(* CODESYS project SPT_Components.library
   Company: Beckhoff Automation LLC
   DefaultNamespace: SPT_Components
   Version: 3.1.1
   Placeholder: SPT Components
   Title: SPT Components

Project tree, tasks and I/O mapping:
  libraries: SPT Base Types, * (Beckhoff Automation LLC); SPT Event Logger, * (Beckhoff Automation LLC); SPT Motion Control, * (Beckhoff Automation LLC); SPT Utilities, * (Beckhoff Automation LLC); Tc2_DataExchange, * (Beckhoff Automation GmbH); Tc2_MC2, * (Beckhoff Automation GmbH); Tc2_Standard, * (Beckhoff Automation GmbH); Tc2_System, * (Beckhoff Automation GmbH); Tc3_EventLogger, * (Beckhoff Automation GmbH); Tc3_Module, * (Beckhoff Automation GmbH); TcUnit, * (www.tcunit.org)
  Axes/
    DUT/
      data type ST_AxisBase_Command
      data type ST_AxisBase_Config
      data type ST_AxisBase_HMI
      data type ST_AxisBase_Status
    function block FB_Component_BasicAxis [ST]: Disable, Enable, Home, Jog, MoveAbsolute, MoveModulo, MoveRelative, MoveVelocity, Reset, Stop, WriteBoolParameter, WriteParameter, Acceleration, Deceleration, Jerk, Velocity, ActualAcceleration, ActualPosition, ActualPositionModulo, ActualTorque, ActualVelocity, PositionLag, SetAcceleration, SetPosition, SetPositionModulo, SetVelocity, Enabled, InPosition, Stopped, Axis, HomeMethod, InhibitFeedNegative, InhibitFeedPositive, Override, ResetMethod, CreateEvents, HMICommunication, Monitoring, CyclicLogic, Initialize
    function block FB_Component_BasicSlaveAxis [ST]: Disable, Enable, Home, Jog, MoveAbsolute, MoveModulo, MoveRelative, MoveVelocity, Reset, Stop, WriteBoolParameter, WriteParameter, Acceleration, Deceleration, Jerk, Velocity, ActualAcceleration, ActualPosition, ActualPositionModulo, ActualTorque, ActualVelocity, PositionLag, SetAcceleration, SetPosition, SetPositionModulo, SetVelocity, Enabled, InPosition, Stopped, Axis, HomeMethod, InhibitFeedNegative, InhibitFeedPositive, Override, ResetMethod, GearIn, GearOut, InGear, Master1, Master2, Master3, Master4, RatioMaster1, RatioMaster2, RatioMaster3, RatioMaster4, CreateEvents, HMICommunication, Monitoring, CyclicLogic, Initialize
    function block FB_Component_CamSlaveAxis [ST]: Disable, Enable, Home, Jog, MoveAbsolute, MoveModulo, MoveRelative, MoveVelocity, Reset, Stop, WriteBoolParameter, WriteParameter, Acceleration, Deceleration, Jerk, Velocity, ActualAcceleration, ActualPosition, ActualPositionModulo, ActualTorque, ActualVelocity, PositionLag, SetAcceleration, SetPosition, SetPositionModulo, SetVelocity, Enabled, InPosition, Stopped, Axis, HomeMethod, InhibitFeedNegative, InhibitFeedPositive, Override, ResetMethod, CamParameters, ChangeMode, FindSlavePos, FindSyncPos, InSync, Master, RunningTable, StartCouple, StartSync, SyncPos, UpdateTable, CreateEvents, HMICommunication, Monitoring, CyclicLogic, Initialize
  GVLs/
    global variables CONSTANTS
  Project Information/
    function F_GetCompany [ST]
    function F_GetTitle [ST]
    function F_GetVersion [ST]
  Sensors/
    DUT/
      data type E_DebounceMode
      data type E_SensorSimulationMode
      data type ST_DigitalSensor_Command
      data type ST_DigitalSensor_Config
      data type ST_DigitalSensor_HMI
      data type ST_DigitalSensor_Status
    function block FB_DigitalSensor [ST]: CyclicLogic, Active, DebounceMode, DebounceTime, Inverted, SimulationInput, SimulationMode, SimulationTimeBase, TimeActive, TimeInactive, HMICommunication, Monitoring, ProcessInput
    interface I_DigitalSensorBase: DebounceMode, DebounceTime, Inverted, SimulationInput, SimulationMode, TimeActive, TimeInactive
  Solenoids/
    DUT/
      data type ST_Cylinder_Command
      data type ST_Cylinder_Config
      data type ST_Cylinder_HMI
      data type ST_Cylinder_Status
    SolenoidBankBase/
      data type E_SolenoidType
      function block FB_SolenoidBankBase [ST]: AddSolenoid, CheckNumber, CreateEvents, CyclicLogic, Initialize, MapIO, Monitoring, Reset
      data type ST_SolenoidBankConfig
    function block FB_DoubleSolenoid [ST]: HardwareInit, HardwareUpdate, RetractOutput
    function block FB_DoubleSolenoidFeedback [ST]: ExtendedInput, Feedback, HardwareInit, RetractedInput
    function block FB_SingleSolenoid [ST]: CreateEvents, HMICommunication, Monitoring, CyclicLogic, Extend, Extended, ExtendOutput, ExtendTime, Retract, Retracted, RetractOutput, RetractTime, Feedback, HardwareInit, HardwareUpdate, Initialize, Reset
    function block FB_SingleSolenoidFeedback [ST]: ExtendedInput, Feedback, HardwareInit, RetractedInput
    interface I_Solenoid: Extend, Extended, ExtendOutput, ExtendTime, Retract, Retracted, RetractOutput, RetractTime
    global variables Parameters_Cylinder
  Testing/
    Axis/
      function block FB_ComponentBasicAxis_Test [ST]: AllowHMI, BlockHMI, Busy, CommandInhibited, Init, MCHaltAlarm, MCHomeAlarm, MCJogAlarm, MCMoveAbsoluteAlarm, MCMoveModulo, MCMoveRelativeAlarm, MCMoveVelocity, MCPowerAlarm, McReadAxisParametersAlarm, MCResetAlarm, McWriteAxisBoolParameterAlarm, McWriteAxisParameterAlarm, NameSetProperty, SimulationCheckAlarm, SimulationSetHMI, SimulationSetProperty
    Solenoids/
      function block FB_DoubleSolenoid_Test [ST]: ExtendEqualsExtendOutputOnRetractOff, RetractEqualsExtendOutputOffRetractOutputOn
      function block FB_SingleSolenoid_Test [ST]: AllowHMI, BlockHMI, Busy, ExtendEqualsExtendedOutputOn, Init, NameSetProperty, RetractEqualsExtendOutputOff, SimulationCheckAlarm, SimulationSetHMI, SimulationSetProperty
      function block FB_SingleSolenoidFeedback_Test [ST]: Extend, ExtendError
    global variables GVL_Testing
    program PRG_TEST [ST]
  Version/
    global variables Global_Version
*)

// Axes/DUT/ST_AxisBase_Command
TYPE ST_AxisBase_Command :
	STRUCT
		JogFast_Forward	 : BOOL;
		JogFast_Backward : BOOL;
		JogSlow_Forward	 : BOOL;
		JogSlow_Backward : BOOL;
	END_STRUCT
END_TYPE

// Axes/DUT/ST_AxisBase_Config
TYPE ST_AxisBase_Config :
	STRUCT
		JogFastVelocity : LREAL;
		JogSlowVelocity : LREAL;
	END_STRUCT
END_TYPE

// Axes/DUT/ST_AxisBase_HMI
TYPE ST_AxisBase_HMI :
	STRUCT
		Config	: ST_AxisBase_Config;
		Command : ST_AxisBase_Command;
		Status	: ST_AxisBase_Status;
	END_STRUCT
END_TYPE

// Axes/DUT/ST_AxisBase_Status
TYPE ST_AxisBase_Status :
	STRUCT
		Enabled				 : BOOL;
		InPosition			 : BOOL;
		Stopped				 : BOOL;
		Coupled				 : BOOL;
		SetPosition			 : LREAL;
		SetPositionModulo	 : LREAL;
		SetVelocity			 : LREAL;
		SetAcceleration		 : LREAL;
		ActualPosition		 : LREAL;
		ActualPositionModulo : LREAL;
		ActualVelocity		 : LREAL;
		ActualAcceleration	 : LREAL;
		ActualTorque		 : LREAL;
		PositionLag			 : LREAL;
	END_STRUCT
END_TYPE

// Sensors/DUT/E_DebounceMode
{attribute 'qualified_only'}
{attribute 'strict'}
TYPE E_DebounceMode : (
		RawInput,
		SimpleFlickerFilter,
		EdgeDetectFilter,
		MovingAverage
	) DINT;
END_TYPE

// Sensors/DUT/E_SensorSimulationMode
{attribute 'qualified_only'}
{attribute 'strict'}
TYPE E_SensorSimulationMode : (
		InputDriven, //Follows the state of the SimulationInput property
		Periodic	 //Follows a 50% duty cycle at the period specified in ms by SimulationInput);
	);
END_TYPE

// Sensors/DUT/ST_DigitalSensor_Command
TYPE ST_DigitalSensor_Command :
	STRUCT
	END_STRUCT
END_TYPE

// Sensors/DUT/ST_DigitalSensor_Config
TYPE ST_DigitalSensor_Config :
	STRUCT
		//Status information
		DebounceMode	   : E_DebounceMode;
		DebounceTime	   : TIME;
		Inverted		   : BOOL;
		SimulationMode	   : E_SensorSimulationMode;
		SimulationTimebase : UINT;
	END_STRUCT
END_TYPE

// Sensors/DUT/ST_DigitalSensor_HMI
TYPE ST_DigitalSensor_HMI :
	STRUCT
		Config	: ST_DigitalSensor_Config;
		Command : ST_DigitalSensor_Command;
		Status	: ST_DigitalSensor_Status;
	END_STRUCT
END_TYPE

// Sensors/DUT/ST_DigitalSensor_Status
TYPE ST_DigitalSensor_Status :
	STRUCT
		Active		 : BOOL;
		TimeActive	 : LREAL;
		TimeInactive : LREAL;
	END_STRUCT
END_TYPE

// Solenoids/DUT/ST_Cylinder_Command
TYPE ST_Cylinder_Command :
	STRUCT
		Extend		: BOOL;
		Retract		: BOOL;
		ExtendTime	: LREAL;
		RetractTime : LREAL;
	END_STRUCT
END_TYPE

// Solenoids/DUT/ST_Cylinder_Config
TYPE ST_Cylinder_Config :
	STRUCT
		ExtendTime	: LREAL;
		RetractTime : LREAL;
	END_STRUCT
END_TYPE

// Solenoids/DUT/ST_Cylinder_HMI
TYPE ST_Cylinder_HMI :
	STRUCT
		Config	: ST_Cylinder_Config;
		Command : ST_Cylinder_Command;
		Status	: ST_Cylinder_Status;
	END_STRUCT
END_TYPE

// Solenoids/DUT/ST_Cylinder_Status
TYPE ST_Cylinder_Status :
	STRUCT
		Extended   : BOOL;
		Retracted  : BOOL;
		Extending  : BOOL;
		Retracting : BOOL;
	END_STRUCT
END_TYPE

// Solenoids/SolenoidBankBase/E_SolenoidType
{attribute 'qualified_only'}
{attribute 'strict'}
TYPE E_SolenoidType : (
		Single,
		Double,
		SingleFeedback,
		DoubleFeedback
	);
END_TYPE

// Solenoids/SolenoidBankBase/ST_SolenoidBankConfig
TYPE ST_SolenoidBankConfig :
	STRUCT
		SolenoidType		 : E_SolenoidType;
		ipSolenoid			 : I_Solenoid;
		SolenoidOutputNumber : UINT;
	END_STRUCT
END_TYPE

// GVLs/CONSTANTS
{attribute 'qualified_only'}
VAR_GLOBAL CONSTANT
	BASIC_AXIS_ALARM_COUNT		 : UINT := 17;
	BASIC_SLAVE_AXIS_ALARM_COUNT : UINT := 3;
	CAM_SLAVE_AXIS_ALARM_COUNT	 : UINT := 9;
END_VAR

// Solenoids/Parameters_Cylinder
{attribute 'qualified_only'}
VAR_GLOBAL CONSTANT
	MAX_NUMBER_OF_SOLENOIDS : UINT := 32;
END_VAR

// Testing/GVL_Testing
{attribute 'qualified_only'}
VAR_GLOBAL
	SingleSolenoidTestsDone : BOOL;
END_VAR

// Version/Global_Version
{attribute 'TcGenerated'}
{attribute 'no-analysis'}
{attribute 'linkalways'}
// This function has been automatically generated from the project information.
VAR_GLOBAL CONSTANT
	{attribute 'const_non_replaced'}
	stLibVersion_SPT_Components : ST_LibVersion := (iMajor := 3, iMinor := 1, iBuild := 1, iRevision := 0, nFlags := 1, sVersion := '3.1.1');
END_VAR

// Axes/FB_Component_BasicAxis
FUNCTION_BLOCK FB_Component_BasicAxis EXTENDS FB_ComponentBase IMPLEMENTS I_BasicAxis
VAR
	BasicAxis				: FB_BasicAxis;
	AxisBase_HMI			: ST_AxisBase_HMI;
	BasicAxisAlarms			: ARRAY[1..CONSTANTS.BASIC_AXIS_ALARM_COUNT] OF FB_TcAlarm;
	HMICommand_BasicAxis_RT : R_TRIG;
END_VAR

// There should be no code in the function block body of I_CyclicFB

METHOD Disable : BOOL
Disable := BasicAxis.Disable();
END_METHOD

METHOD Enable : BOOL
Enable := BasicAxis.Enable();
END_METHOD

METHOD Home : BOOL
Home := BasicAxis.Home();
END_METHOD

METHOD Jog : BOOL
VAR_INPUT
	JogFW	 : BOOL;
	JogBW	 : BOOL;
	JogMode	 : E_JogMode;
	Position : LREAL;
END_VAR
Jog := BasicAxis.Jog(JogFW,
					 JogBW,
					 JogMode,
					 Position);
END_METHOD

METHOD MoveAbsolute : BOOL
VAR_INPUT
	Position	  : LREAL;
	AbortPrevious : BOOL;
END_VAR
MoveAbsolute := BasicAxis.MoveAbsolute(Position, AbortPrevious);
END_METHOD

METHOD MoveModulo : BOOL
VAR_INPUT
	Position	  : LREAL;
	Direction	  : MC_Direction;
	AbortPrevious : BOOL;
END_VAR
MoveModulo := BasicAxis.MoveModulo(Position, Direction, AbortPrevious);
END_METHOD

METHOD MoveRelative : BOOL
VAR_INPUT
	Distance	  : LREAL;
	AbortPrevious : BOOL;
END_VAR
MoveRelative := BasicAxis.MoveRelative(Distance, AbortPrevious);
END_METHOD

METHOD MoveVelocity : BOOL
VAR_INPUT
	Velocity	  : LREAL;
	AbortPrevious : BOOL;
END_VAR
MoveVelocity := BasicAxis.MoveVelocity(Velocity, AbortPrevious);
END_METHOD

METHOD Reset : BOOL
Reset := FALSE;
SUPER^.Reset();
IF BasicAxis.ResetMethod = 0 THEN
	RETURN;
ELSIF BasicAxis.HomeMethod = 0 THEN
	RETURN;
ELSE
	IF (BasicAxis.ResetMethod.Error AND BasicAxis.ResetPreviouslyErrored) AND BasicAxisAlarms[E_BasicAxis.ResetError].bRaised THEN
		BasicAxisAlarms[E_BasicAxis.ResetError].Clear(0, 0);
	END_IF

	IF (BasicAxis.HomeMethod.Error AND BasicAxis.HomePreviouslyErrored) AND BasicAxisAlarms[E_BasicAxis.HomeError].bRaised THEN
		BasicAxisAlarms[E_BasicAxis.HomeError].Clear(0, 0);
	END_IF

	IF BasicAxis.Reset() THEN
		_Error	 := FALSE;
		_ErrorID := 0;
		Reset	 := TRUE;
	END_IF
END_IF
END_METHOD

METHOD Stop : BOOL
Stop := BasicAxis.Stop();
END_METHOD

METHOD WriteBoolParameter : BOOL
VAR_INPUT
	ParameterNumber : MC_AxisParameter;
	Value			: BOOL;
END_VAR
WriteBoolParameter := BasicAxis.WriteBoolParameter(ParameterNumber, Value);
END_METHOD

METHOD WriteParameter : BOOL
VAR_INPUT
	ParameterNumber : MC_AxisParameter;
	Value			: LREAL;
END_VAR
WriteParameter := BasicAxis.WriteParameter(ParameterNumber, Value);
END_METHOD

PROPERTY Acceleration : LREAL
GET
Acceleration := BasicAxis.Acceleration;
END_GET
SET
BasicAxis.Acceleration := Acceleration;
END_SET
END_PROPERTY

PROPERTY Deceleration : LREAL
GET
Deceleration := BasicAxis.Deceleration;
END_GET
SET
BasicAxis.Deceleration := Deceleration;
END_SET
END_PROPERTY

PROPERTY Jerk : LREAL
GET
Jerk := BasicAxis.Jerk;
END_GET
SET
BasicAxis.Jerk := Jerk;
END_SET
END_PROPERTY

PROPERTY Velocity : LREAL
GET
Velocity := BasicAxis.Velocity;
END_GET
SET
BasicAxis.Velocity := Velocity;
END_SET
END_PROPERTY

PROPERTY ActualAcceleration : LREAL
GET
ActualAcceleration := BasicAxis.ActualAcceleration;
END_GET
END_PROPERTY

PROPERTY ActualPosition : LREAL
GET
ActualPosition := BasicAxis.ActualPosition;
END_GET
END_PROPERTY

PROPERTY ActualPositionModulo : LREAL
GET
ActualPositionModulo := BasicAxis.ActualPositionModulo;
END_GET
END_PROPERTY

PROPERTY ActualTorque : LREAL
GET
ActualTorque := BasicAxis.ActualTorque;
END_GET
END_PROPERTY

PROPERTY ActualVelocity : LREAL
GET
ActualVelocity := BasicAxis.ActualVelocity;
END_GET
END_PROPERTY

PROPERTY PositionLag : LREAL
GET
PositionLag := BasicAxis.PositionLag;
END_GET
END_PROPERTY

PROPERTY SetAcceleration : LREAL
GET
SetAcceleration := BasicAxis.SetAcceleration;
END_GET
END_PROPERTY

PROPERTY SetPosition : LREAL
GET
SetPosition := BasicAxis.SetPosition;
END_GET
END_PROPERTY

PROPERTY SetPositionModulo : LREAL
GET
SetPositionModulo := BasicAxis.SetPositionModulo;
END_GET
END_PROPERTY

PROPERTY SetVelocity : LREAL
GET
SetVelocity := BasicAxis.SetVelocity;
END_GET
END_PROPERTY

PROPERTY Enabled : BOOL
GET
Enabled := BasicAxis.Enabled;
END_GET
END_PROPERTY

PROPERTY InPosition : BOOL
GET
InPosition := BasicAxis.InPosition;
END_GET
END_PROPERTY

PROPERTY Stopped : BOOL
GET
Stopped := BasicAxis.Stopped;
END_GET
END_PROPERTY

{attribute 'analysis' := '-29'}
PROPERTY Axis : REFERENCE TO AXIS_REF
GET
Axis REF= BasicAxis.Axis;
END_GET
END_PROPERTY

PROPERTY HomeMethod : I_MotionSequence
SET
BasicAxis.HomeMethod := HomeMethod;
END_SET
END_PROPERTY

PROPERTY InhibitFeedNegative : BOOL
SET
BasicAxis.InhibitFeedNegative := InhibitFeedNegative;
END_SET
END_PROPERTY

PROPERTY InhibitFeedPositive : BOOL
SET
BasicAxis.InhibitFeedPositive := InhibitFeedPositive;
END_SET
END_PROPERTY

PROPERTY Override : LREAL
GET
Override := BasicAxis.Override;
END_GET
SET
IF Override >= 0 AND Override <= 100 THEN
	BasicAxis.Override := Override;
END_IF
END_SET
END_PROPERTY

PROPERTY ResetMethod : I_MotionSequence
SET
BasicAxis.ResetMethod := ResetMethod;
END_SET
END_PROPERTY

{attribute 'call_after_online_change_slot' := '<slot>'}
METHOD PROTECTED CreateEvents
VAR
	Temp : STRING;
END_VAR
Temp := CONCAT(CONCAT(CONCAT('Axis ', ': '), Name),
			   ' '); //Creates a utility string for alarms and other messaging that reads (example text) - "Module 10 - Main Casepacker" to be followed by the alarm or message info

F_CreateAllEventsInClass(Alarms		:= BasicAxisAlarms,
						 ClassSize	:= SIZEOF(TC_EVENTS.BasicAxis),
						 pInitEvent := ADR(TC_EVENTS.BasicAxis.InitReferenceEvent),
						 Prefix		:= Name);

SUPER^.CreateEvents();
END_METHOD

METHOD PROTECTED HMICommunication
//Extend this method in extended FBs to communicate specific implementation data
SUPER^.HMICommunication();

//Process HMI requests

//Replace 'FALSE' below with further momentary commands (myCommand XOR myOtherCommand XOR...)
HMICommand_BasicAxis_RT(CLK := (ComponentBase_HMI.Status.HMIControlAvailable AND NOT HMICommandActive_Base));

//Signal to FB_ComponentBase that a command is active
HMICommandActive_Descendant := ComponentBase_HMI.Status.HMIControlAvailable AND
							   (AxisBase_HMI.Command.JogFast_Backward OR AxisBase_HMI.Command.JogFast_Forward OR AxisBase_HMI.Command.JogSlow_Forward OR AxisBase_HMI.Command.JogSlow_Backward);

//Process HMI requests
IF HMICommand_BasicAxis_RT.Q THEN //If a request has been issued by the HMI, and a previous request has not just finished being processed
END_IF

IF ComponentBase_HMI.Status.HMIControlAvailable AND NOT HMICommand_BasicAxis_RT.Q THEN
	IF AxisBase_HMI.Command.JogSlow_Forward THEN
		BasicAxis.Jog(AxisBase_HMI.Command.JogSlow_Forward,
					  FALSE,
					  E_JogMode.MC_JOGMODE_STANDARD_SLOW,
					  0.0);
	ELSIF AxisBase_HMI.Command.JogSlow_Backward THEN
		BasicAxis.Jog(FALSE,
					  AxisBase_HMI.Command.JogSlow_Backward,
					  E_JogMode.MC_JOGMODE_STANDARD_SLOW,
					  0.0);
	ELSIF AxisBase_HMI.Command.JogFast_Forward THEN
		BasicAxis.Jog(AxisBase_HMI.Command.JogFast_Forward,
					  FALSE,
					  E_JogMode.MC_JOGMODE_STANDARD_FAST,
					  0.0);
	ELSIF AxisBase_HMI.Command.JogFast_Backward THEN
		BasicAxis.Jog(FALSE,
					  AxisBase_HMI.Command.JogFast_Backward,
					  E_JogMode.MC_JOGMODE_STANDARD_FAST,
					  0.0);
	ELSE
		BasicAxis.Jog(FALSE,
					  FALSE,
					  E_JogMode.MC_JOGMODE_STANDARD_SLOW,
					  0.0);
	END_IF
END_IF

//Update HMI status info
AxisBase_HMI.Status.Enabled				 := BasicAxis.Enabled;
AxisBase_HMI.Status.InPosition			 := BasicAxis.InPosition;
AxisBase_HMI.Status.Stopped				 := BasicAxis.Stopped;
AxisBase_HMI.Status.Coupled				 := FALSE;
AxisBase_HMI.Status.SetPosition			 := BasicAxis.SetPosition;
AxisBase_HMI.Status.SetPositionModulo	 := BasicAxis.SetPositionModulo;
AxisBase_HMI.Status.SetVelocity			 := BasicAxis.SetVelocity;
AxisBase_HMI.Status.SetAcceleration		 := BasicAxis.SetAcceleration;
AxisBase_HMI.Status.ActualPosition		 := BasicAxis.ActualPosition;
AxisBase_HMI.Status.ActualPositionModulo := BasicAxis.ActualPositionModulo;
AxisBase_HMI.Status.ActualVelocity		 := BasicAxis.ActualVelocity;
AxisBase_HMI.Status.ActualAcceleration	 := BasicAxis.ActualAcceleration;
AxisBase_HMI.Status.ActualTorque		 := BasicAxis.ActualTorque;
AxisBase_HMI.Status.PositionLag			 := BasicAxis.PositionLag;
END_METHOD

METHOD PROTECTED Monitoring
SUPER^.Monitoring();

//ErrorID 2 - MC_Power
IF BasicAxis.MCPower.Error AND NOT BasicAxisAlarms[E_BasicAxis.PowerError].bRaised THEN
	RaiseAlarmWithStrings(Alarm := BasicAxisAlarms[E_BasicAxis.PowerError], UDINT_TO_STRING(BasicAxis.ErrorID), '');
ELSIF NOT BasicAxis.MCPower.Error AND BasicAxisAlarms[E_BasicAxis.PowerError].bRaised THEN
	BasicAxisAlarms[E_BasicAxis.PowerError].Clear(0, 0);
END_IF

//ErrorID 3 - MC_Reset (or other reset method)
IF BasicAxis.ResetMethod <> 0 THEN
	IF (BasicAxis.ResetMethod.Error AND NOT BasicAxis.ResetPreviouslyErrored) AND NOT BasicAxisAlarms[E_BasicAxis.ResetError].bRaised THEN
		RaiseAlarmWithStrings(Alarm := BasicAxisAlarms[E_BasicAxis.ResetError], UDINT_TO_STRING(BasicAxis.ResetMethod.ErrorID), '');
	ELSIF NOT BasicAxis.ResetMethod.Error AND BasicAxisAlarms[E_BasicAxis.ResetError].bRaised THEN
		BasicAxisAlarms[E_BasicAxis.ResetError].Clear(0, 0);
	END_IF
END_IF

//ErrorID 4 - MC_Halt
IF BasicAxis.MCHalt.Error AND NOT BasicAxisAlarms[E_BasicAxis.HaltError].bRaised THEN
	RaiseAlarmWithStrings(Alarm := BasicAxisAlarms[E_BasicAxis.HaltError], UDINT_TO_STRING(BasicAxis.MCHalt.ErrorID), '');
ELSIF NOT BasicAxis.MCHalt.Error AND BasicAxisAlarms[E_BasicAxis.HaltError].bRaised THEN
	BasicAxisAlarms[E_BasicAxis.HaltError].Clear(0, 0);
END_IF

//ErrorID 5 - MC_Stop **NOT IMPLEMENTED**

//ErrorID 6 - MC_Home (or other home method)
IF BasicAxis.HomeMethod <> 0 THEN
	IF (BasicAxis.HomeMethod.Error AND NOT BasicAxis.HomePreviouslyErrored) AND NOT BasicAxisAlarms[E_BasicAxis.HomeError].bRaised THEN
		RaiseAlarmWithStrings(Alarm := BasicAxisAlarms[E_BasicAxis.HomeError], UDINT_TO_STRING(BasicAxis.HomeMethod.ErrorID), '');
	ELSIF NOT BasicAxis.HomeMethod.Error AND BasicAxisAlarms[E_BasicAxis.HomeError].bRaised THEN
		BasicAxisAlarms[E_BasicAxis.HomeError].Clear(0, 0);
	END_IF
END_IF

//ErrorID 7 - MC_Jog 
IF BasicAxis.MCJog.Error AND NOT BasicAxisAlarms[E_BasicAxis.JogError].bRaised THEN
	RaiseAlarmWithStrings(Alarm := BasicAxisAlarms[E_BasicAxis.JogError], UDINT_TO_STRING(BasicAxis.MCJog.ErrorID), '');
ELSIF NOT BasicAxis.MCJog.Error AND BasicAxisAlarms[E_BasicAxis.JogError].bRaised THEN
	BasicAxisAlarms[E_BasicAxis.JogError].Clear(0, 0);
END_IF

//ErrorID 8 - MC_MoveAbsolute
IF BasicAxis.MCMoveAbsolute <> 0 THEN
	IF BasicAxis.MCMoveAbsolute^.Error AND NOT BasicAxisAlarms[E_BasicAxis.MoveAbsoluteError].bRaised THEN
		RaiseAlarmWithStrings(Alarm := BasicAxisAlarms[E_BasicAxis.MoveAbsoluteError], UDINT_TO_STRING(BasicAxis.MCMoveAbsolute^.ErrorID), '');
	ELSIF NOT BasicAxis.MCMoveAbsolute^.Error AND BasicAxisAlarms[E_BasicAxis.MoveAbsoluteError].bRaised THEN
		BasicAxisAlarms[E_BasicAxis.MoveAbsoluteError].Clear(0, 0);
	END_IF
END_IF

//ErrorID 9 - MC_MoveRelative
IF BasicAxis.MCMoveRelative <> 0 THEN
	IF BasicAxis.MCMoveRelative^.Error AND NOT BasicAxisAlarms[E_BasicAxis.MoveRelativeError].bRaised THEN
		RaiseAlarmWithStrings(Alarm := BasicAxisAlarms[E_BasicAxis.MoveRelativeError], UDINT_TO_STRING(BasicAxis.MCMoveRelative^.ErrorID), '');
	ELSIF NOT BasicAxis.MCMoveRelative^.Error AND BasicAxisAlarms[E_BasicAxis.MoveRelativeError].bRaised THEN
		BasicAxisAlarms[E_BasicAxis.MoveRelativeError].Clear(0, 0);
	END_IF
END_IF

//ErrorID 10 - MC_MoveVelocity
IF BasicAxis.MCMoveVelocity <> 0 THEN
	IF BasicAxis.MCMoveVelocity^.Error AND NOT BasicAxisAlarms[E_BasicAxis.MoveVelocityError].bRaised THEN
		RaiseAlarmWithStrings(Alarm := BasicAxisAlarms[E_BasicAxis.MoveVelocityError], UDINT_TO_STRING(BasicAxis.MCMoveVelocity^.ErrorID), '');
	ELSIF NOT BasicAxis.MCMoveVelocity^.Error AND BasicAxisAlarms[E_BasicAxis.MoveVelocityError].bRaised THEN
		BasicAxisAlarms[E_BasicAxis.MoveVelocityError].Clear(0, 0);
	END_IF
END_IF

//ErrorID 11 - MC_MoveModulo
IF BasicAxis.MCMoveModulo <> 0 THEN
	IF BasicAxis.MCMoveModulo^.Error AND NOT BasicAxisAlarms[E_BasicAxis.MoveModuloError].bRaised THEN
		RaiseAlarmWithStrings(Alarm := BasicAxisAlarms[E_BasicAxis.MoveModuloError], UDINT_TO_STRING(BasicAxis.MCMoveModulo^.ErrorID), '');
	ELSIF NOT BasicAxis.MCMoveModulo^.Error AND BasicAxisAlarms[E_BasicAxis.MoveModuloError].bRaised THEN
		BasicAxisAlarms[E_BasicAxis.MoveModuloError].Clear(0, 0);
	END_IF
END_IF

//ErrorID 12 - MC_ReadParameterSet
IF BasicAxis.MCReadParameterSet.Error AND NOT BasicAxisAlarms[E_BasicAxis.ReadParameterSetError].bRaised THEN
	RaiseAlarmWithStrings(Alarm := BasicAxisAlarms[E_BasicAxis.ReadParameterSetError], UDINT_TO_STRING(BasicAxis.MCReadParameterSet.ErrorID), '');
ELSIF NOT BasicAxis.MCReadParameterSet.Error AND BasicAxisAlarms[E_BasicAxis.ReadParameterSetError].bRaised THEN
	BasicAxisAlarms[E_BasicAxis.ReadParameterSetError].Clear(0, 0);
END_IF

//ErrorID 13 - MC_WriteParameter
IF BasicAxis.MCWriteParameter.Error AND NOT BasicAxisAlarms[E_BasicAxis.WriteParameterError].bRaised THEN
	RaiseAlarmWithStrings(Alarm := BasicAxisAlarms[E_BasicAxis.WriteParameterError], UDINT_TO_STRING(BasicAxis.MCWriteParameter.ErrorID), '');
ELSIF NOT BasicAxis.MCWriteParameter.Error AND BasicAxisAlarms[E_BasicAxis.WriteParameterError].bRaised THEN
	BasicAxisAlarms[E_BasicAxis.WriteParameterError].Clear(0, 0);
END_IF

//ErrorID 14 - MC_WriteBoolParameter
IF BasicAxis.MCWriteBoolParameter.Error AND NOT BasicAxisAlarms[E_BasicAxis.WriteBoolParameterError].bRaised THEN
	RaiseAlarmWithStrings(Alarm := BasicAxisAlarms[E_BasicAxis.WriteBoolParameterError], UDINT_TO_STRING(BasicAxis.MCWriteBoolParameter.ErrorID), '');
ELSIF NOT BasicAxis.MCWriteBoolParameter.Error AND BasicAxisAlarms[E_BasicAxis.WriteBoolParameterError].bRaised THEN
	BasicAxisAlarms[E_BasicAxis.WriteBoolParameterError].Clear(0, 0);
END_IF

//ErrorID 15 - Command While Inhibited (WARNING)
IF ((BasicAxis.Override <= 0) AND _Busy) AND NOT BasicAxisAlarms[E_BasicAxis.CommandWhileInhibited].bRaised THEN
	RaiseAlarm(Alarm := BasicAxisAlarms[E_BasicAxis.CommandWhileInhibited]);
ELSIF NOT ((BasicAxis.Override <= 0) AND _Busy) AND BasicAxisAlarms[E_BasicAxis.CommandWhileInhibited].bRaised THEN
	BasicAxisAlarms[E_BasicAxis.CommandWhileInhibited].Clear(0, 0);
END_IF

//ErrorID 16 - NC Axis Error
IF BasicAxis.Axis.Status.Error AND NOT BasicAxisAlarms[E_BasicAxis.AxisError].bRaised THEN
	RaiseAlarmWithStrings(Alarm := BasicAxisAlarms[E_BasicAxis.AxisError], UDINT_TO_STRING(BasicAxis.Axis.Status.ErrorID), '');
ELSIF NOT BasicAxis.Axis.Status.Error AND BasicAxisAlarms[E_BasicAxis.AxisError].bRaised THEN
	BasicAxisAlarms[E_BasicAxis.AxisError].Clear(0, 0);
END_IF

//ErrorID 17 - Hardware Error **TODO**
_CurrentAlarmSeverity := F_GetMaxSeverityRaised(Alarms := BasicAxisAlarms, CurrentSeverity := CurrentAlarmSeverity);
END_METHOD

METHOD CyclicLogic
SUPER^.CyclicLogic();
BasicAxis.CyclicLogic();
_Busy	 := BasicAxis.Busy;
_Error	 := BasicAxis.Error;
_ErrorID := BasicAxis.ErrorID;
END_METHOD

//! @summary Basic component initialization logic
METHOD PROTECTED Initialize : BOOL;

//! @description This method is called by <c>CyclicLogic()</c> as required
Initialize := FALSE;
IF NOT BasicAxis.InitComplete THEN
	RETURN;
END_IF

Initialize := SUPER^.Initialize();
END_METHOD

END_FUNCTION_BLOCK

// Axes/FB_Component_BasicSlaveAxis
FUNCTION_BLOCK FB_Component_BasicSlaveAxis EXTENDS FB_ComponentBase IMPLEMENTS I_BasicSlaveAxis
VAR
	BasicSlaveAxis				 : FB_BasicSlaveAxis;
	AxisBase_HMI				 : ST_AxisBase_HMI;
	BasicAxisAlarms				 : ARRAY[1..CONSTANTS.BASIC_AXIS_ALARM_COUNT] OF FB_TcAlarm;
	BasicSlaveAxisAlarms		 : ARRAY[1..CONSTANTS.BASIC_SLAVE_AXIS_ALARM_COUNT] OF FB_TcAlarm;
	HMICommand_BasicSlaveAxis_RT : R_TRIG;
END_VAR

// There should be no code in the function block body of I_CyclicFB

METHOD Disable : BOOL
Disable := BasicSlaveAxis.Disable();
END_METHOD

METHOD Enable : BOOL
Enable := BasicSlaveAxis.Enable();
END_METHOD

METHOD Home : BOOL
Home := BasicSlaveAxis.Home();
END_METHOD

METHOD Jog : BOOL
VAR_INPUT
	JogFW	 : BOOL;
	JogBW	 : BOOL;
	JogMode	 : E_JogMode;
	Position : LREAL;
END_VAR
Jog := BasicSlaveAxis.Jog(JogFW,
						  JogBW,
						  JogMode,
						  Position);
END_METHOD

METHOD MoveAbsolute : BOOL
VAR_INPUT
	Position	  : LREAL;
	AbortPrevious : BOOL;
END_VAR
MoveAbsolute := BasicSlaveAxis.MoveAbsolute(Position, AbortPrevious);
END_METHOD

METHOD MoveModulo : BOOL
VAR_INPUT
	Position	  : LREAL;
	Direction	  : MC_Direction;
	AbortPrevious : BOOL;
END_VAR
MoveModulo := BasicSlaveAxis.MoveModulo(Position, Direction, AbortPrevious);
END_METHOD

METHOD MoveRelative : BOOL
VAR_INPUT
	Distance	  : LREAL;
	AbortPrevious : BOOL;
END_VAR
MoveRelative := BasicSlaveAxis.MoveRelative(Distance, AbortPrevious);
END_METHOD

METHOD MoveVelocity : BOOL
VAR_INPUT
	Velocity	  : LREAL;
	AbortPrevious : BOOL;
END_VAR
MoveVelocity := BasicSlaveAxis.MoveVelocity(Velocity, AbortPrevious);
END_METHOD

METHOD Reset : BOOL
SUPER^.Reset();
IF BasicSlaveAxis.ResetMethod = 0 THEN
	RETURN;
ELSE
	IF (BasicSlaveAxis.ResetMethod.Error AND BasicSlaveAxis.ResetPreviouslyErrored) AND BasicAxisAlarms[E_BasicAxis.ResetError].bRaised THEN
		BasicAxisAlarms[E_BasicAxis.ResetError].Clear(0, 0);
	END_IF

	IF (BasicSlaveAxis.HomeMethod.Error AND BasicSlaveAxis.HomePreviouslyErrored) AND BasicAxisAlarms[E_BasicAxis.HomeError].bRaised THEN
		BasicAxisAlarms[E_BasicAxis.HomeError].Clear(0, 0);
	END_IF

	IF BasicSlaveAxis.Reset() THEN
		_Error	 := FALSE;
		_ErrorID := 0;
		Reset	 := TRUE;
	END_IF
END_IF
END_METHOD

METHOD Stop : BOOL
Stop := BasicSlaveAxis.Stop();
END_METHOD

METHOD WriteBoolParameter : BOOL
VAR_INPUT
	ParameterNumber : MC_AxisParameter;
	Value			: BOOL;
END_VAR
WriteBoolParameter := BasicSlaveAxis.WriteBoolParameter(ParameterNumber, Value);
END_METHOD

METHOD WriteParameter : BOOL
VAR_INPUT
	ParameterNumber : MC_AxisParameter;
	Value			: LREAL;
END_VAR
WriteParameter := BasicSlaveAxis.WriteParameter(ParameterNumber, Value);
END_METHOD

PROPERTY Acceleration : LREAL
GET
Acceleration := BasicSlaveAxis.Acceleration;
END_GET
SET
BasicSlaveAxis.Acceleration := Acceleration;
END_SET
END_PROPERTY

PROPERTY Deceleration : LREAL
GET
Deceleration := BasicSlaveAxis.Deceleration;
END_GET
SET
BasicSlaveAxis.Deceleration := Deceleration;
END_SET
END_PROPERTY

PROPERTY Jerk : LREAL
GET
Jerk := BasicSlaveAxis.Jerk;
END_GET
SET
BasicSlaveAxis.Jerk := Jerk;
END_SET
END_PROPERTY

PROPERTY Velocity : LREAL
GET
Velocity := BasicSlaveAxis.Velocity;
END_GET
SET
BasicSlaveAxis.Velocity := Velocity;
END_SET
END_PROPERTY

PROPERTY ActualAcceleration : LREAL
GET
ActualAcceleration := BasicSlaveAxis.ActualAcceleration;
END_GET
END_PROPERTY

PROPERTY ActualPosition : LREAL
GET
ActualPosition := BasicSlaveAxis.ActualPosition;
END_GET
END_PROPERTY

PROPERTY ActualPositionModulo : LREAL
GET
ActualPositionModulo := BasicSlaveAxis.ActualPositionModulo;
END_GET
END_PROPERTY

PROPERTY ActualTorque : LREAL
GET
ActualTorque := BasicSlaveAxis.ActualTorque;
END_GET
END_PROPERTY

PROPERTY ActualVelocity : LREAL
GET
ActualVelocity := BasicSlaveAxis.ActualVelocity;
END_GET
END_PROPERTY

PROPERTY PositionLag : LREAL
GET
PositionLag := BasicSlaveAxis.PositionLag;
END_GET
END_PROPERTY

PROPERTY SetAcceleration : LREAL
GET
SetAcceleration := BasicSlaveAxis.SetAcceleration;
END_GET
END_PROPERTY

PROPERTY SetPosition : LREAL
GET
SetPosition := BasicSlaveAxis.SetPosition;
END_GET
END_PROPERTY

PROPERTY SetPositionModulo : LREAL
GET
SetPositionModulo := BasicSlaveAxis.SetPositionModulo;
END_GET
END_PROPERTY

PROPERTY SetVelocity : LREAL
GET
SetVelocity := BasicSlaveAxis.SetVelocity;
END_GET
END_PROPERTY

PROPERTY Enabled : BOOL
GET
Enabled := BasicSlaveAxis.Enabled;
END_GET
END_PROPERTY

PROPERTY InPosition : BOOL
GET
InPosition := BasicSlaveAxis.InPosition;
END_GET
END_PROPERTY

PROPERTY Stopped : BOOL
GET
Stopped := BasicSlaveAxis.Stopped;
END_GET
END_PROPERTY

PROPERTY Axis : REFERENCE TO AXIS_REF
GET
Axis REF= BasicSlaveAxis.Axis;
END_GET
END_PROPERTY

PROPERTY HomeMethod : I_MotionSequence
SET
BasicSlaveAxis.HomeMethod := HomeMethod;
END_SET
END_PROPERTY

PROPERTY InhibitFeedNegative : BOOL
SET
BasicSlaveAxis.InhibitFeedNegative := InhibitFeedNegative;
END_SET
END_PROPERTY

PROPERTY InhibitFeedPositive : BOOL
SET
BasicSlaveAxis.InhibitFeedPositive := InhibitFeedPositive;
END_SET
END_PROPERTY

PROPERTY Override : LREAL
GET
Override := BasicSlaveAxis.Override;
END_GET
SET
IF Override >= 0 AND Override <= 100 THEN
	BasicSlaveAxis.Override := Override;
END_IF
END_SET
END_PROPERTY

PROPERTY ResetMethod : I_MotionSequence
SET
BasicSlaveAxis.ResetMethod := ResetMethod;
END_SET
END_PROPERTY

METHOD PUBLIC GearIn : BOOL
VAR_INPUT
END_VAR
GearIn := BasicSlaveAxis.GearIn();
END_METHOD

METHOD GearOut : BOOL
GearOut := BasicSlaveAxis.GearOut();
END_METHOD

PROPERTY InGear : BOOL
GET
InGear := BasicSlaveAxis.InGear;
END_GET
END_PROPERTY

PROPERTY Master1 : REFERENCE TO AXIS_REF
GET
IF __ISVALIDREF(BasicSlaveAxis.Master1) THEN
	Master1 REF= BasicSlaveAxis.Master1;
END_IF
END_GET
SET
BasicSlaveAxis.Master1 REF= Master1;
END_SET
END_PROPERTY

PROPERTY Master2 : REFERENCE TO AXIS_REF
GET
IF __ISVALIDREF(BasicSlaveAxis.Master2) THEN
	Master2 REF= BasicSlaveAxis.Master2;
END_IF
END_GET
SET
BasicSlaveAxis.Master2 REF= Master2;
END_SET
END_PROPERTY

PROPERTY Master3 : REFERENCE TO AXIS_REF
GET
IF __ISVALIDREF(BasicSlaveAxis.Master3) THEN
	Master3 REF= BasicSlaveAxis.Master3;
END_IF
END_GET
SET
BasicSlaveAxis.Master3 REF= Master3;
END_SET
END_PROPERTY

PROPERTY Master4 : REFERENCE TO AXIS_REF
GET
IF __ISVALIDREF(BasicSlaveAxis.Master4) THEN
	Master4 REF= BasicSlaveAxis.Master4;
END_IF
END_GET
SET
BasicSlaveAxis.Master4 REF= Master4;
END_SET
END_PROPERTY

PROPERTY RatioMaster1 : LREAL
GET
RatioMaster1 := BasicSlaveAxis.RatioMaster1;
END_GET
SET
BasicSlaveAxis.RatioMaster1 := RatioMaster1;
END_SET
END_PROPERTY

PROPERTY RatioMaster2 : LREAL
GET
RatioMaster2 := BasicSlaveAxis.RatioMaster2;
END_GET
SET
BasicSlaveAxis.RatioMaster2 := RatioMaster2;
END_SET
END_PROPERTY

PROPERTY RatioMaster3 : LREAL
GET
RatioMaster3 := BasicSlaveAxis.RatioMaster3;
END_GET
SET
BasicSlaveAxis.RatioMaster3 := RatioMaster3;
END_SET
END_PROPERTY

PROPERTY RatioMaster4 : LREAL
GET
RatioMaster4 := BasicSlaveAxis.RatioMaster4;
END_GET
SET
BasicSlaveAxis.RatioMaster4 := RatioMaster4;
END_SET
END_PROPERTY

{attribute 'call_after_online_change_slot' := '<slot>'}
METHOD PROTECTED CreateEvents
VAR
	Temp : STRING;
END_VAR
Temp := CONCAT(CONCAT(CONCAT('Axis ', ': '), Name),
			   ' '); //Creates a utility string for alarms and other messaging that reads (example text) - "Module 10 - Main Casepacker" to be followed by the alarm or message info

F_CreateAllEventsInClass(Alarms		:= BasicAxisAlarms,
						 ClassSize	:= SIZEOF(TC_EVENTS.BasicAxis),
						 pInitEvent := ADR(TC_EVENTS.BasicAxis.InitReferenceEvent),
						 Prefix		:= Name);

F_CreateAllEventsInClass(Alarms		:= BasicSlaveAxisAlarms,
						 ClassSize	:= SIZEOF(TC_EVENTS.BasicSlaveAxis),
						 pInitEvent := ADR(TC_EVENTS.BasicSlaveAxis.InitReferenceEvent),
						 Prefix		:= Name);

SUPER^.CreateEvents();
END_METHOD

METHOD PROTECTED HMICommunication
//Extend this method in extended FBs to communicate specific implementation data
SUPER^.HMICommunication();

//Process HMI requests

//Replace 'FALSE' below with further momentary commands (myCommand XOR myOtherCommand XOR...)
HMICommand_BasicSlaveAxis_RT(CLK := (ComponentBase_HMI.Status.HMIControlAvailable AND NOT HMICommandActive_Base) AND (FALSE));

//Signal to FB_ComponentBase that a command is active
HMICommandActive_Descendant := ComponentBase_HMI.Status.HMIControlAvailable AND
							   (AxisBase_HMI.Command.JogFast_Backward OR AxisBase_HMI.Command.JogFast_Forward OR AxisBase_HMI.Command.JogSlow_Forward OR AxisBase_HMI.Command.JogSlow_Backward);

IF HMICommand_BasicSlaveAxis_RT.Q THEN
	;
END_IF

//Process HMI requests
IF HMICommand_BasicSlaveAxis_RT.Q THEN //If a request has been issued by the HMI, and a previous request has not just finished being processed

	//	IF AxisBaseHMI.Command.xxx THEN

	//		Enabled := TRUE;

	//	END_IF
END_IF

IF ComponentBase_HMI.Status.HMIControlAvailable AND NOT HMICommand_BasicSlaveAxis_RT.Q THEN
	IF AxisBase_HMI.Command.JogSlow_Forward THEN
		BasicSlaveAxis.Jog(AxisBase_HMI.Command.JogSlow_Forward,
						   FALSE,
						   E_JogMode.MC_JOGMODE_STANDARD_SLOW,
						   0.0);
	ELSIF AxisBase_HMI.Command.JogSlow_Backward THEN
		BasicSlaveAxis.Jog(FALSE,
						   AxisBase_HMI.Command.JogSlow_Backward,
						   E_JogMode.MC_JOGMODE_STANDARD_SLOW,
						   0.0);
	ELSIF AxisBase_HMI.Command.JogFast_Forward THEN
		BasicSlaveAxis.Jog(AxisBase_HMI.Command.JogFast_Forward,
						   FALSE,
						   E_JogMode.MC_JOGMODE_STANDARD_FAST,
						   0.0);
	ELSIF AxisBase_HMI.Command.JogFast_Backward THEN
		BasicSlaveAxis.Jog(FALSE,
						   AxisBase_HMI.Command.JogFast_Backward,
						   E_JogMode.MC_JOGMODE_STANDARD_FAST,
						   0.0);
	ELSE
		BasicSlaveAxis.Jog(FALSE,
						   FALSE,
						   E_JogMode.MC_JOGMODE_STANDARD_SLOW,
						   0.0);
	END_IF
END_IF

//Update HMI status info
AxisBase_HMI.Status.Enabled				 := BasicSlaveAxis.Enabled;
AxisBase_HMI.Status.InPosition			 := BasicSlaveAxis.InPosition;
AxisBase_HMI.Status.Stopped				 := BasicSlaveAxis.Stopped;
AxisBase_HMI.Status.Coupled				 := BasicSlaveAxis.InGear;
AxisBase_HMI.Status.SetPosition			 := BasicSlaveAxis.SetPosition;
AxisBase_HMI.Status.SetPositionModulo	 := BasicSlaveAxis.SetPositionModulo;
AxisBase_HMI.Status.SetVelocity			 := BasicSlaveAxis.SetVelocity;
AxisBase_HMI.Status.SetAcceleration		 := BasicSlaveAxis.SetAcceleration;
AxisBase_HMI.Status.ActualPosition		 := BasicSlaveAxis.ActualPosition;
AxisBase_HMI.Status.ActualPositionModulo := BasicSlaveAxis.ActualPositionModulo;
AxisBase_HMI.Status.ActualVelocity		 := BasicSlaveAxis.ActualVelocity;
AxisBase_HMI.Status.ActualAcceleration	 := BasicSlaveAxis.ActualAcceleration;
AxisBase_HMI.Status.ActualTorque		 := BasicSlaveAxis.ActualTorque;
AxisBase_HMI.Status.PositionLag			 := BasicSlaveAxis.PositionLag;
END_METHOD

METHOD PROTECTED Monitoring
SUPER^.Monitoring();

(* Basic Axis Alarms *)

//ErrorID 2 - MC_Power
IF BasicSlaveAxis.MCPower.Error AND NOT BasicAxisAlarms[E_BasicAxis.PowerError].bRaised THEN
	RaiseAlarmWithStrings(Alarm := BasicAxisAlarms[E_BasicAxis.PowerError], UDINT_TO_STRING(BasicSlaveAxis.ErrorID), '');
ELSIF NOT BasicSlaveAxis.MCPower.Error AND BasicAxisAlarms[E_BasicAxis.PowerError].bRaised THEN
	BasicAxisAlarms[E_BasicAxis.PowerError].Clear(0, 0);
END_IF

//ErrorID 3 - MC_Reset (or other reset method)
IF BasicSlaveAxis.ResetMethod <> 0 THEN
	IF (BasicSlaveAxis.ResetMethod.Error AND NOT BasicSlaveAxis.ResetPreviouslyErrored) AND NOT BasicAxisAlarms[E_BasicAxis.ResetError].bRaised THEN
		RaiseAlarmWithStrings(Alarm := BasicAxisAlarms[E_BasicAxis.ResetError], UDINT_TO_STRING(BasicSlaveAxis.ResetMethod.ErrorID), '');
	ELSIF NOT BasicSlaveAxis.ResetMethod.Error AND BasicAxisAlarms[E_BasicAxis.ResetError].bRaised THEN
		BasicAxisAlarms[E_BasicAxis.ResetError].Clear(0, 0);
	END_IF
END_IF

//ErrorID 4 - MC_Halt
IF BasicSlaveAxis.MCHalt.Error AND NOT BasicAxisAlarms[E_BasicAxis.HaltError].bRaised THEN
	RaiseAlarmWithStrings(Alarm := BasicAxisAlarms[E_BasicAxis.HaltError], UDINT_TO_STRING(BasicSlaveAxis.MCHalt.ErrorID), '');
ELSIF NOT BasicSlaveAxis.MCHalt.Error AND BasicAxisAlarms[E_BasicAxis.HaltError].bRaised THEN
	BasicAxisAlarms[E_BasicAxis.HaltError].Clear(0, 0);
END_IF

//ErrorID 5 - MC_Stop **NOT IMPLEMENTED**

//ErrorID 6 - MC_Home (or other home method)
IF BasicSlaveAxis.HomeMethod <> 0 THEN
	IF (BasicSlaveAxis.HomeMethod.Error AND NOT BasicSlaveAxis.HomePreviouslyErrored) AND NOT BasicAxisAlarms[E_BasicAxis.HomeError].bRaised THEN
		RaiseAlarmWithStrings(Alarm := BasicAxisAlarms[E_BasicAxis.HomeError], UDINT_TO_STRING(BasicSlaveAxis.HomeMethod.ErrorID), '');
	ELSIF NOT BasicSlaveAxis.HomeMethod.Error AND BasicAxisAlarms[E_BasicAxis.HomeError].bRaised THEN
		BasicAxisAlarms[E_BasicAxis.HomeError].Clear(0, 0);
	END_IF
END_IF

//ErrorID 7 - MC_Jog 
IF BasicSlaveAxis.MCJog.Error AND NOT BasicAxisAlarms[E_BasicAxis.JogError].bRaised THEN
	RaiseAlarmWithStrings(Alarm := BasicAxisAlarms[E_BasicAxis.JogError], UDINT_TO_STRING(BasicSlaveAxis.MCJog.ErrorID), '');
ELSIF NOT BasicSlaveAxis.MCJog.Error AND BasicAxisAlarms[E_BasicAxis.JogError].bRaised THEN
	BasicAxisAlarms[E_BasicAxis.JogError].Clear(0, 0);
END_IF

//ErrorID 8 - MC_MoveAbsolute
IF BasicSlaveAxis.MCMoveAbsolute <> 0 THEN
	IF BasicSlaveAxis.MCMoveAbsolute^.Error AND NOT BasicAxisAlarms[E_BasicAxis.MoveAbsoluteError].bRaised THEN
		RaiseAlarmWithStrings(Alarm := BasicAxisAlarms[E_BasicAxis.MoveAbsoluteError], UDINT_TO_STRING(BasicSlaveAxis.MCMoveAbsolute^.ErrorID), '');
	ELSIF NOT BasicSlaveAxis.MCMoveAbsolute^.Error AND BasicAxisAlarms[E_BasicAxis.MoveAbsoluteError].bRaised THEN
		BasicAxisAlarms[E_BasicAxis.MoveAbsoluteError].Clear(0, 0);
	END_IF
END_IF

//ErrorID 9 - MC_MoveRelative
IF BasicSlaveAxis.MCMoveRelative <> 0 THEN
	IF BasicSlaveAxis.MCMoveRelative^.Error AND NOT BasicAxisAlarms[E_BasicAxis.MoveRelativeError].bRaised THEN
		RaiseAlarmWithStrings(Alarm := BasicAxisAlarms[E_BasicAxis.MoveRelativeError], UDINT_TO_STRING(BasicSlaveAxis.MCMoveRelative^.ErrorID), '');
	ELSIF NOT BasicSlaveAxis.MCMoveRelative^.Error AND BasicAxisAlarms[E_BasicAxis.MoveRelativeError].bRaised THEN
		BasicAxisAlarms[E_BasicAxis.MoveRelativeError].Clear(0, 0);
	END_IF
END_IF

//ErrorID 10 - MC_MoveVelocity
IF BasicSlaveAxis.MCMoveVelocity <> 0 THEN
	IF BasicSlaveAxis.MCMoveVelocity^.Error AND NOT BasicAxisAlarms[E_BasicAxis.MoveVelocityError].bRaised THEN
		RaiseAlarmWithStrings(Alarm := BasicAxisAlarms[E_BasicAxis.MoveVelocityError], UDINT_TO_STRING(BasicSlaveAxis.MCMoveVelocity^.ErrorID), '');
	ELSIF NOT BasicSlaveAxis.MCMoveVelocity^.Error AND BasicAxisAlarms[E_BasicAxis.MoveVelocityError].bRaised THEN
		BasicAxisAlarms[E_BasicAxis.MoveVelocityError].Clear(0, 0);
	END_IF
END_IF

//ErrorID 11 - MC_MoveModulo
IF BasicSlaveAxis.MCMoveModulo <> 0 THEN
	IF BasicSlaveAxis.MCMoveModulo^.Error AND NOT BasicAxisAlarms[E_BasicAxis.MoveModuloError].bRaised THEN
		RaiseAlarmWithStrings(Alarm := BasicAxisAlarms[E_BasicAxis.MoveModuloError], UDINT_TO_STRING(BasicSlaveAxis.MCMoveModulo^.ErrorID), '');
	ELSIF NOT BasicSlaveAxis.MCMoveModulo^.Error AND BasicAxisAlarms[E_BasicAxis.MoveModuloError].bRaised THEN
		BasicAxisAlarms[E_BasicAxis.MoveModuloError].Clear(0, 0);
	END_IF
END_IF

//ErrorID 12 - MC_ReadParameterSet
IF BasicSlaveAxis.MCReadParameterSet.Error AND NOT BasicAxisAlarms[E_BasicAxis.ReadParameterSetError].bRaised THEN
	RaiseAlarmWithStrings(Alarm := BasicAxisAlarms[E_BasicAxis.ReadParameterSetError], UDINT_TO_STRING(BasicSlaveAxis.MCReadParameterSet.ErrorID), '');
ELSIF NOT BasicSlaveAxis.MCReadParameterSet.Error AND BasicAxisAlarms[E_BasicAxis.ReadParameterSetError].bRaised THEN
	BasicAxisAlarms[E_BasicAxis.ReadParameterSetError].Clear(0, 0);
END_IF

//ErrorID 13 - MC_WriteParameter
IF BasicSlaveAxis.MCWriteParameter.Error AND NOT BasicAxisAlarms[E_BasicAxis.WriteParameterError].bRaised THEN
	RaiseAlarmWithStrings(Alarm := BasicAxisAlarms[E_BasicAxis.WriteParameterError], UDINT_TO_STRING(BasicSlaveAxis.MCWriteParameter.ErrorID), '');
ELSIF NOT BasicSlaveAxis.MCWriteParameter.Error AND BasicAxisAlarms[E_BasicAxis.WriteParameterError].bRaised THEN
	BasicAxisAlarms[E_BasicAxis.WriteParameterError].Clear(0, 0);
END_IF

//ErrorID 14 - MC_WriteBoolParameter
IF BasicSlaveAxis.MCWriteBoolParameter.Error AND NOT BasicAxisAlarms[E_BasicAxis.WriteBoolParameterError].bRaised THEN
	RaiseAlarmWithStrings(Alarm := BasicAxisAlarms[E_BasicAxis.WriteBoolParameterError], UDINT_TO_STRING(BasicSlaveAxis.MCWriteBoolParameter.ErrorID), '');
ELSIF NOT BasicSlaveAxis.MCWriteBoolParameter.Error AND BasicAxisAlarms[E_BasicAxis.WriteBoolParameterError].bRaised THEN
	BasicAxisAlarms[E_BasicAxis.WriteBoolParameterError].Clear(0, 0);
END_IF

//ErrorID 15 - Command While Inhibited (WARNING)
IF ((BasicSlaveAxis.Override <= 0) AND _Busy) AND NOT BasicAxisAlarms[E_BasicAxis.CommandWhileInhibited].bRaised THEN
	RaiseAlarm(Alarm := BasicAxisAlarms[E_BasicAxis.CommandWhileInhibited]);
ELSIF NOT ((BasicSlaveAxis.Override <= 0) AND _Busy) AND BasicAxisAlarms[E_BasicAxis.CommandWhileInhibited].bRaised THEN
	BasicAxisAlarms[E_BasicAxis.CommandWhileInhibited].Clear(0, 0);
END_IF

//ErrorID 16 - NC Axis Error
IF BasicSlaveAxis.Axis.Status.Error AND NOT BasicAxisAlarms[E_BasicAxis.AxisError].bRaised THEN
	RaiseAlarmWithStrings(Alarm := BasicAxisAlarms[E_BasicAxis.AxisError], UDINT_TO_STRING(BasicSlaveAxis.Axis.Status.ErrorID), '');
ELSIF NOT BasicSlaveAxis.Axis.Status.Error AND BasicAxisAlarms[E_BasicAxis.AxisError].bRaised THEN
	BasicAxisAlarms[E_BasicAxis.AxisError].Clear(0, 0);
END_IF

//ErrorID 17 - Hardware Error **TODO**

(* Basic Slave Axis Alarms *)

//ErrorID 2 - MC_GearInMultimaster
IF BasicSlaveAxis.MCGearInMultimaster.Error AND NOT BasicAxisAlarms[E_BasicSlaveAxis.GearInMultimasterError].bRaised THEN
	RaiseAlarmWithStrings(Alarm := BasicSlaveAxisAlarms[E_BasicSlaveAxis.GearInMultimasterError], UDINT_TO_STRING(BasicSlaveAxis.MCGearInMultimaster.ErrorID), '');
ELSIF NOT BasicSlaveAxis.MCGearInMultimaster.Error AND BasicSlaveAxisAlarms[E_BasicSlaveAxis.GearInMultimasterError].bRaised THEN
	BasicSlaveAxisAlarms[E_BasicSlaveAxis.GearInMultimasterError].Clear(0, 0);
END_IF

//ErrorID 3 - MC_GearOut
IF BasicSlaveAxis.MCGearOut.Error AND NOT BasicAxisAlarms[E_BasicSlaveAxis.GearOutError].bRaised THEN
	RaiseAlarmWithStrings(Alarm := BasicSlaveAxisAlarms[E_BasicSlaveAxis.GearOutError], UDINT_TO_STRING(BasicSlaveAxis.MCGearOut.ErrorID), '');
ELSIF NOT BasicSlaveAxis.MCGearOut.Error AND BasicSlaveAxisAlarms[E_BasicSlaveAxis.GearOutError].bRaised THEN
	BasicSlaveAxisAlarms[E_BasicSlaveAxis.GearOutError].Clear(0, 0);
END_IF

_CurrentAlarmSeverity := F_GetMaxSeverityRaised(Alarms := BasicAxisAlarms, CurrentSeverity := CurrentAlarmSeverity);
_CurrentAlarmSeverity := F_GetMaxSeverityRaised(Alarms := BasicSlaveAxisAlarms, CurrentSeverity := CurrentAlarmSeverity);
END_METHOD

METHOD CyclicLogic
SUPER^.CyclicLogic();
BasicSlaveAxis.CyclicLogic();
_Busy	 := BasicSlaveAxis.Busy;
_Error	 := BasicSlaveAxis.Error;
_ErrorID := BasicSlaveAxis.ErrorID;
END_METHOD

//! @summary Basic component initialization logic
METHOD PROTECTED Initialize : BOOL;

//! @description This method is called by <c>CyclicLogic()</c> as required
IF NOT BasicSlaveAxis.InitComplete THEN
	RETURN;
END_IF

Initialize := SUPER^.Initialize();
END_METHOD

END_FUNCTION_BLOCK

// Axes/FB_Component_CamSlaveAxis
FUNCTION_BLOCK FB_Component_CamSlaveAxis EXTENDS FB_ComponentBase IMPLEMENTS I_CamSlaveAxis
VAR
	CamSlaveAxis			   : FB_CamSlaveAxis;
	AxisBase_HMI			   : ST_AxisBase_HMI;
	BasicAxisAlarms			   : ARRAY[1..CONSTANTS.BASIC_AXIS_ALARM_COUNT] OF FB_TcAlarm;
	CamSlaveAxisAlarms		   : ARRAY[1..CONSTANTS.CAM_SLAVE_AXIS_ALARM_COUNT] OF FB_TcAlarm;
	HMICommand_CamSlaveAxis_RT : R_TRIG;
END_VAR

// There should be no code in the function block body of I_CyclicFB

METHOD Disable : BOOL
Disable := CamSlaveAxis.Disable();
END_METHOD

METHOD Enable : BOOL
Enable := CamSlaveAxis.Enable();
END_METHOD

METHOD Home : BOOL
Home := CamSlaveAxis.Home();
END_METHOD

METHOD Jog : BOOL
VAR_INPUT
	JogFW	 : BOOL;
	JogBW	 : BOOL;
	JogMode	 : E_JogMode;
	Position : LREAL;
END_VAR
Jog := CamSlaveAxis.Jog(JogFW,
						JogBW,
						JogMode,
						Position);
END_METHOD

METHOD MoveAbsolute : BOOL
VAR_INPUT
	Position	  : LREAL;
	AbortPrevious : BOOL;
END_VAR
MoveAbsolute := CamSlaveAxis.MoveAbsolute(Position, AbortPrevious);
END_METHOD

METHOD MoveModulo : BOOL
VAR_INPUT
	Position	  : LREAL;
	Direction	  : MC_Direction;
	AbortPrevious : BOOL;
END_VAR
MoveModulo := CamSlaveAxis.MoveModulo(Position, Direction, AbortPrevious);
END_METHOD

METHOD MoveRelative : BOOL
VAR_INPUT
	Distance	  : LREAL;
	AbortPrevious : BOOL;
END_VAR
MoveRelative := CamSlaveAxis.MoveRelative(Distance, AbortPrevious);
END_METHOD

METHOD MoveVelocity : BOOL
VAR_INPUT
	Velocity	  : LREAL;
	AbortPrevious : BOOL;
END_VAR
MoveVelocity := CamSlaveAxis.MoveVelocity(Velocity, AbortPrevious);
END_METHOD

METHOD Reset : BOOL
SUPER^.Reset();
IF CamSlaveAxis.ResetMethod = 0 THEN
	RETURN;
ELSE
	IF (CamSlaveAxis.ResetMethod.Error AND CamSlaveAxis.ResetPreviouslyErrored) AND BasicAxisAlarms[E_BasicAxis.ResetError].bRaised THEN
		BasicAxisAlarms[E_BasicAxis.ResetError].Clear(0, 0);
	END_IF

	IF (CamSlaveAxis.HomeMethod.Error AND CamSlaveAxis.HomePreviouslyErrored) AND BasicAxisAlarms[E_BasicAxis.HomeError].bRaised THEN
		BasicAxisAlarms[E_BasicAxis.HomeError].Clear(0, 0);
	END_IF

	IF CamSlaveAxis.Reset() THEN
		_Error	 := FALSE;
		_ErrorID := 0;
		Reset	 := TRUE;
	END_IF
END_IF
END_METHOD

METHOD Stop : BOOL
Stop := CamSlaveAxis.Stop();
END_METHOD

METHOD WriteBoolParameter : BOOL
VAR_INPUT
	ParameterNumber : MC_AxisParameter;
	Value			: BOOL;
END_VAR
WriteBoolParameter := CamSlaveAxis.WriteBoolParameter(ParameterNumber, Value);
END_METHOD

METHOD WriteParameter : BOOL
VAR_INPUT
	ParameterNumber : MC_AxisParameter;
	Value			: LREAL;
END_VAR
WriteParameter := CamSlaveAxis.WriteParameter(ParameterNumber, Value);
END_METHOD

PROPERTY Acceleration : LREAL
GET
Acceleration := CamSlaveAxis.Acceleration;
END_GET
SET
CamSlaveAxis.Acceleration := Acceleration;
END_SET
END_PROPERTY

PROPERTY Deceleration : LREAL
GET
Deceleration := CamSlaveAxis.Deceleration;
END_GET
SET
CamSlaveAxis.Deceleration := Deceleration;
END_SET
END_PROPERTY

PROPERTY Jerk : LREAL
GET
Jerk := CamSlaveAxis.Jerk;
END_GET
SET
CamSlaveAxis.Jerk := Jerk;
END_SET
END_PROPERTY

PROPERTY Velocity : LREAL
GET
Velocity := CamSlaveAxis.Velocity;
END_GET
SET
CamSlaveAxis.Velocity := Velocity;
END_SET
END_PROPERTY

PROPERTY ActualAcceleration : LREAL
GET
ActualAcceleration := CamSlaveAxis.ActualAcceleration;
END_GET
END_PROPERTY

PROPERTY ActualPosition : LREAL
GET
ActualPosition := CamSlaveAxis.ActualPosition;
END_GET
END_PROPERTY

PROPERTY ActualPositionModulo : LREAL
GET
ActualPositionModulo := CamSlaveAxis.ActualPositionModulo;
END_GET
END_PROPERTY

PROPERTY ActualTorque : LREAL
GET
ActualTorque := CamSlaveAxis.ActualTorque;
END_GET
END_PROPERTY

PROPERTY ActualVelocity : LREAL
GET
ActualVelocity := CamSlaveAxis.ActualVelocity;
END_GET
END_PROPERTY

PROPERTY PositionLag : LREAL
GET
PositionLag := CamSlaveAxis.PositionLag;
END_GET
END_PROPERTY

PROPERTY SetAcceleration : LREAL
GET
SetAcceleration := CamSlaveAxis.SetAcceleration;
END_GET
END_PROPERTY

PROPERTY SetPosition : LREAL
GET
SetPosition := CamSlaveAxis.SetPosition;
END_GET
END_PROPERTY

PROPERTY SetPositionModulo : LREAL
GET
SetPositionModulo := CamSlaveAxis.SetPositionModulo;
END_GET
END_PROPERTY

PROPERTY SetVelocity : LREAL
GET
SetVelocity := CamSlaveAxis.SetVelocity;
END_GET
END_PROPERTY

PROPERTY Enabled : BOOL
GET
Enabled := CamSlaveAxis.Enabled;
END_GET
END_PROPERTY

PROPERTY InPosition : BOOL
GET
InPosition := CamSlaveAxis.InPosition;
END_GET
END_PROPERTY

PROPERTY Stopped : BOOL
GET
Stopped := CamSlaveAxis.Stopped;
END_GET
END_PROPERTY

PROPERTY Axis : REFERENCE TO AXIS_REF
GET
Axis REF= CamSlaveAxis.Axis;
END_GET
END_PROPERTY

PROPERTY HomeMethod : I_MotionSequence
SET
CamSlaveAxis.HomeMethod := HomeMethod;
END_SET
END_PROPERTY

PROPERTY InhibitFeedNegative : BOOL
SET
CamSlaveAxis.InhibitFeedNegative := InhibitFeedNegative;
END_SET
END_PROPERTY

PROPERTY InhibitFeedPositive : BOOL
SET
CamSlaveAxis.InhibitFeedPositive := InhibitFeedPositive;
END_SET
END_PROPERTY

PROPERTY Override : LREAL
GET
Override := CamSlaveAxis.Override;
END_GET
SET
IF Override >= 0 AND Override <= 100 THEN
	CamSlaveAxis.Override := Override;
END_IF
END_SET
END_PROPERTY

PROPERTY ResetMethod : I_MotionSequence
SET
CamSlaveAxis.ResetMethod := ResetMethod;
END_SET
END_PROPERTY

PROPERTY CamParameters : REFERENCE TO ST_CamParameters
GET
IF __ISVALIDREF(CamSlaveAxis._CamParameters) THEN
	CamParameters REF= CamSlaveAxis._CamParameters;
END_IF
END_GET
SET
CamSlaveAxis.CamParameters REF= CamParameters;
END_SET
END_PROPERTY

METHOD ChangeMode : BOOL
VAR_INPUT
END_VAR
ChangeMode := CamSlaveAxis.ChangeMode();
END_METHOD

METHOD FindSlavePos : BOOL
VAR_INPUT
END_VAR
FindSlavePos := CamSlaveAxis.FindSlavePos();
END_METHOD

METHOD FindSyncPos : BOOL
VAR_INPUT
END_VAR
FindSyncPos := CamSlaveAxis.FindSyncPos();
END_METHOD

PROPERTY InSync : BOOL
GET
InSync := CamSlaveAxis._InSync;
END_GET
END_PROPERTY

PROPERTY Master : REFERENCE TO Tc2_MC2.AXIS_REF
GET
IF __ISVALIDREF(CamSlaveAxis.Master) THEN
	Master REF= CamSlaveAxis.Master;
END_IF
END_GET
SET
CamSlaveAxis.Master REF= Master;
END_SET
END_PROPERTY

PROPERTY RunningTable : UDINT
GET
RunningTable := CamSlaveAxis._RunningTable;
END_GET
END_PROPERTY

METHOD StartCouple : BOOL
VAR_INPUT
END_VAR
StartCouple := CamSlaveAxis.StartCouple();
END_METHOD

METHOD StartSync : BOOL
VAR_INPUT
END_VAR
StartSync := CamSlaveAxis.StartSync();
END_METHOD

PROPERTY SyncPos : LREAL
GET
SyncPos := CamSlaveAxis._SyncPos;
END_GET
END_PROPERTY

METHOD UpdateTable : BOOL
VAR_INPUT
END_VAR
UpdateTable := CamSlaveAxis.UpdateTable();
END_METHOD

{attribute 'call_after_online_change_slot' := '<slot>'}
METHOD PROTECTED CreateEvents
VAR
	Temp : STRING;
END_VAR
Temp := CONCAT(CONCAT(CONCAT('Axis ', ': '), Name),
			   ' '); //Creates a utility string for alarms and other messaging that reads (example text) - "Module 10 - Main Casepacker" to be followed by the alarm or message info

F_CreateAllEventsInClass(Alarms		:= BasicAxisAlarms,
						 ClassSize	:= SIZEOF(TC_EVENTS.BasicAxis),
						 pInitEvent := ADR(TC_EVENTS.BasicAxis.InitReferenceEvent),
						 Prefix		:= Name);

F_CreateAllEventsInClass(Alarms		:= CamSlaveAxisAlarms,
						 ClassSize	:= SIZEOF(TC_EVENTS.CamSlaveAxis),
						 pInitEvent := ADR(TC_EVENTS.CamSlaveAxis.InitReferenceEvent),
						 Prefix		:= Name);

SUPER^.CreateEvents();
END_METHOD

METHOD PROTECTED HMICommunication
//Extend this method in extended FBs to communicate specific implementation data
SUPER^.HMICommunication();

//Process HMI requests

//Replace 'FALSE' below with further momentary commands (myCommand XOR myOtherCommand XOR...)
HMICommand_CamSlaveAxis_RT(CLK := (ComponentBase_HMI.Status.HMIControlAvailable AND NOT HMICommandActive_Base) AND (FALSE));

//Signal to FB_ComponentBase that a command is active
HMICommandActive_Descendant := ComponentBase_HMI.Status.HMIControlAvailable AND
							   (AxisBase_HMI.Command.JogFast_Backward OR AxisBase_HMI.Command.JogFast_Forward OR AxisBase_HMI.Command.JogSlow_Forward OR AxisBase_HMI.Command.JogSlow_Backward);

IF HMICommand_CamSlaveAxis_RT.Q THEN
	;
END_IF

//Process HMI requests
IF HMICommand_CamSlaveAxis_RT.Q THEN //If a request has been issued by the HMI, and a previous request has not just finished being processed

	//	IF AxisBaseHMI.Command.xxx THEN

	//		Enabled := TRUE;

	//	END_IF
END_IF

IF ComponentBase_HMI.Status.HMIControlAvailable AND NOT HMICommand_CamSlaveAxis_RT.Q THEN
	IF AxisBase_HMI.Command.JogSlow_Forward THEN
		CamSlaveAxis.Jog(AxisBase_HMI.Command.JogSlow_Forward,
						 FALSE,
						 E_JogMode.MC_JOGMODE_STANDARD_SLOW,
						 0.0);
	ELSIF AxisBase_HMI.Command.JogSlow_Backward THEN
		CamSlaveAxis.Jog(FALSE,
						 AxisBase_HMI.Command.JogSlow_Backward,
						 E_JogMode.MC_JOGMODE_STANDARD_SLOW,
						 0.0);
	ELSIF AxisBase_HMI.Command.JogFast_Forward THEN
		CamSlaveAxis.Jog(AxisBase_HMI.Command.JogFast_Forward,
						 FALSE,
						 E_JogMode.MC_JOGMODE_STANDARD_FAST,
						 0.0);
	ELSIF AxisBase_HMI.Command.JogFast_Backward THEN
		CamSlaveAxis.Jog(FALSE,
						 AxisBase_HMI.Command.JogFast_Backward,
						 E_JogMode.MC_JOGMODE_STANDARD_FAST,
						 0.0);
	ELSE
		CamSlaveAxis.Jog(FALSE,
						 FALSE,
						 E_JogMode.MC_JOGMODE_STANDARD_SLOW,
						 0.0);
	END_IF
END_IF

//Update HMI status info
AxisBase_HMI.Status.Enabled				 := CamSlaveAxis.Enabled;
AxisBase_HMI.Status.InPosition			 := CamSlaveAxis.InPosition;
AxisBase_HMI.Status.Stopped				 := CamSlaveAxis.Stopped;
AxisBase_HMI.Status.Coupled				 := CamSlaveAxis.InSync;
AxisBase_HMI.Status.SetPosition			 := CamSlaveAxis.SetPosition;
AxisBase_HMI.Status.SetPositionModulo	 := CamSlaveAxis.SetPositionModulo;
AxisBase_HMI.Status.SetVelocity			 := CamSlaveAxis.SetVelocity;
AxisBase_HMI.Status.SetAcceleration		 := CamSlaveAxis.SetAcceleration;
AxisBase_HMI.Status.ActualPosition		 := CamSlaveAxis.ActualPosition;
AxisBase_HMI.Status.ActualPositionModulo := CamSlaveAxis.ActualPositionModulo;
AxisBase_HMI.Status.ActualVelocity		 := CamSlaveAxis.ActualVelocity;
AxisBase_HMI.Status.ActualAcceleration	 := CamSlaveAxis.ActualAcceleration;
AxisBase_HMI.Status.ActualTorque		 := CamSlaveAxis.ActualTorque;
AxisBase_HMI.Status.PositionLag			 := CamSlaveAxis.PositionLag;
END_METHOD

METHOD PROTECTED Monitoring
SUPER^.Monitoring();

(* Basic Axis Alarms *)

//ErrorID 2 - MC_Power
IF CamSlaveAxis.MCPower.Error AND NOT BasicAxisAlarms[E_BasicAxis.PowerError].bRaised THEN
	RaiseAlarmWithStrings(Alarm := BasicAxisAlarms[E_BasicAxis.PowerError], UDINT_TO_STRING(CamSlaveAxis.ErrorID), '');
ELSIF NOT CamSlaveAxis.MCPower.Error AND BasicAxisAlarms[E_BasicAxis.PowerError].bRaised THEN
	BasicAxisAlarms[E_BasicAxis.PowerError].Clear(0, 0);
END_IF

//ErrorID 3 - MC_Reset (or other reset method)
IF CamSlaveAxis.ResetMethod <> 0 THEN
	IF (CamSlaveAxis.ResetMethod.Error AND NOT CamSlaveAxis.ResetPreviouslyErrored) AND NOT BasicAxisAlarms[E_BasicAxis.ResetError].bRaised THEN
		RaiseAlarmWithStrings(Alarm := BasicAxisAlarms[E_BasicAxis.ResetError], UDINT_TO_STRING(CamSlaveAxis.ResetMethod.ErrorID), '');
	ELSIF NOT CamSlaveAxis.ResetMethod.Error AND BasicAxisAlarms[E_BasicAxis.ResetError].bRaised THEN
		BasicAxisAlarms[E_BasicAxis.ResetError].Clear(0, 0);
	END_IF
END_IF

//ErrorID 4 - MC_Halt
IF CamSlaveAxis.MCHalt.Error AND NOT BasicAxisAlarms[E_BasicAxis.HaltError].bRaised THEN
	RaiseAlarmWithStrings(Alarm := BasicAxisAlarms[E_BasicAxis.HaltError], UDINT_TO_STRING(CamSlaveAxis.MCHalt.ErrorID), '');
ELSIF NOT CamSlaveAxis.MCHalt.Error AND BasicAxisAlarms[E_BasicAxis.HaltError].bRaised THEN
	BasicAxisAlarms[E_BasicAxis.HaltError].Clear(0, 0);
END_IF

//ErrorID 5 - MC_Stop **NOT IMPLEMENTED**

//ErrorID 6 - MC_Home (or other home method)
IF CamSlaveAxis.HomeMethod <> 0 THEN
	IF (CamSlaveAxis.HomeMethod.Error AND NOT CamSlaveAxis.HomePreviouslyErrored) AND NOT BasicAxisAlarms[E_BasicAxis.HomeError].bRaised THEN
		RaiseAlarmWithStrings(Alarm := BasicAxisAlarms[E_BasicAxis.HomeError], UDINT_TO_STRING(CamSlaveAxis.HomeMethod.ErrorID), '');
	ELSIF NOT CamSlaveAxis.HomeMethod.Error AND BasicAxisAlarms[E_BasicAxis.HomeError].bRaised THEN
		BasicAxisAlarms[E_BasicAxis.HomeError].Clear(0, 0);
	END_IF
END_IF

//ErrorID 7 - MC_Jog 
IF CamSlaveAxis.MCJog.Error AND NOT BasicAxisAlarms[E_BasicAxis.JogError].bRaised THEN
	RaiseAlarmWithStrings(Alarm := BasicAxisAlarms[E_BasicAxis.JogError], UDINT_TO_STRING(CamSlaveAxis.MCJog.ErrorID), '');
ELSIF NOT CamSlaveAxis.MCJog.Error AND BasicAxisAlarms[E_BasicAxis.JogError].bRaised THEN
	BasicAxisAlarms[E_BasicAxis.JogError].Clear(0, 0);
END_IF

//ErrorID 8 - MC_MoveAbsolute
IF CamSlaveAxis.MCMoveAbsolute <> 0 THEN
	IF CamSlaveAxis.MCMoveAbsolute^.Error AND NOT BasicAxisAlarms[E_BasicAxis.MoveAbsoluteError].bRaised THEN
		RaiseAlarmWithStrings(Alarm := BasicAxisAlarms[E_BasicAxis.MoveAbsoluteError], UDINT_TO_STRING(CamSlaveAxis.MCMoveAbsolute^.ErrorID), '');
	ELSIF NOT CamSlaveAxis.MCMoveAbsolute^.Error AND BasicAxisAlarms[E_BasicAxis.MoveAbsoluteError].bRaised THEN
		BasicAxisAlarms[E_BasicAxis.MoveAbsoluteError].Clear(0, 0);
	END_IF
END_IF

//ErrorID 9 - MC_MoveRelative
IF CamSlaveAxis.MCMoveRelative <> 0 THEN
	IF CamSlaveAxis.MCMoveRelative^.Error AND NOT BasicAxisAlarms[E_BasicAxis.MoveRelativeError].bRaised THEN
		RaiseAlarmWithStrings(Alarm := BasicAxisAlarms[E_BasicAxis.MoveRelativeError], UDINT_TO_STRING(CamSlaveAxis.MCMoveRelative^.ErrorID), '');
	ELSIF NOT CamSlaveAxis.MCMoveRelative^.Error AND BasicAxisAlarms[E_BasicAxis.MoveRelativeError].bRaised THEN
		BasicAxisAlarms[E_BasicAxis.MoveRelativeError].Clear(0, 0);
	END_IF
END_IF

//ErrorID 10 - MC_MoveVelocity
IF CamSlaveAxis.MCMoveVelocity <> 0 THEN
	IF CamSlaveAxis.MCMoveVelocity^.Error AND NOT BasicAxisAlarms[E_BasicAxis.MoveVelocityError].bRaised THEN
		RaiseAlarmWithStrings(Alarm := BasicAxisAlarms[E_BasicAxis.MoveVelocityError], UDINT_TO_STRING(CamSlaveAxis.MCMoveVelocity^.ErrorID), '');
	ELSIF NOT CamSlaveAxis.MCMoveVelocity^.Error AND BasicAxisAlarms[E_BasicAxis.MoveVelocityError].bRaised THEN
		BasicAxisAlarms[E_BasicAxis.MoveVelocityError].Clear(0, 0);
	END_IF
END_IF

//ErrorID 11 - MC_MoveModulo
IF CamSlaveAxis.MCMoveModulo <> 0 THEN
	IF CamSlaveAxis.MCMoveModulo^.Error AND NOT BasicAxisAlarms[E_BasicAxis.MoveModuloError].bRaised THEN
		RaiseAlarmWithStrings(Alarm := BasicAxisAlarms[E_BasicAxis.MoveModuloError], UDINT_TO_STRING(CamSlaveAxis.MCMoveModulo^.ErrorID), '');
	ELSIF NOT CamSlaveAxis.MCMoveModulo^.Error AND BasicAxisAlarms[E_BasicAxis.MoveModuloError].bRaised THEN
		BasicAxisAlarms[E_BasicAxis.MoveModuloError].Clear(0, 0);
	END_IF
END_IF

//ErrorID 12 - MC_ReadParameterSet
IF CamSlaveAxis.MCReadParameterSet.Error AND NOT BasicAxisAlarms[E_BasicAxis.ReadParameterSetError].bRaised THEN
	RaiseAlarmWithStrings(Alarm := BasicAxisAlarms[E_BasicAxis.ReadParameterSetError], UDINT_TO_STRING(CamSlaveAxis.MCReadParameterSet.ErrorID), '');
ELSIF NOT CamSlaveAxis.MCReadParameterSet.Error AND BasicAxisAlarms[E_BasicAxis.ReadParameterSetError].bRaised THEN
	BasicAxisAlarms[E_BasicAxis.ReadParameterSetError].Clear(0, 0);
END_IF

//ErrorID 13 - MC_WriteParameter
IF CamSlaveAxis.MCWriteParameter.Error AND NOT BasicAxisAlarms[E_BasicAxis.WriteParameterError].bRaised THEN
	RaiseAlarmWithStrings(Alarm := BasicAxisAlarms[E_BasicAxis.WriteParameterError], UDINT_TO_STRING(CamSlaveAxis.MCWriteParameter.ErrorID), '');
ELSIF NOT CamSlaveAxis.MCWriteParameter.Error AND BasicAxisAlarms[E_BasicAxis.WriteParameterError].bRaised THEN
	BasicAxisAlarms[E_BasicAxis.WriteParameterError].Clear(0, 0);
END_IF

//ErrorID 14 - MC_WriteBoolParameter
IF CamSlaveAxis.MCWriteBoolParameter.Error AND NOT BasicAxisAlarms[E_BasicAxis.WriteBoolParameterError].bRaised THEN
	RaiseAlarmWithStrings(Alarm := BasicAxisAlarms[E_BasicAxis.WriteBoolParameterError], UDINT_TO_STRING(CamSlaveAxis.MCWriteBoolParameter.ErrorID), '');
ELSIF NOT CamSlaveAxis.MCWriteBoolParameter.Error AND BasicAxisAlarms[E_BasicAxis.WriteBoolParameterError].bRaised THEN
	BasicAxisAlarms[E_BasicAxis.WriteBoolParameterError].Clear(0, 0);
END_IF

//ErrorID 15 - Command While Inhibited (WARNING)
IF ((CamSlaveAxis.Override <= 0) AND _Busy) AND NOT BasicAxisAlarms[E_BasicAxis.CommandWhileInhibited].bRaised THEN
	RaiseAlarm(Alarm := BasicAxisAlarms[E_BasicAxis.CommandWhileInhibited]);
ELSIF NOT ((CamSlaveAxis.Override <= 0) AND _Busy) AND BasicAxisAlarms[E_BasicAxis.CommandWhileInhibited].bRaised THEN
	BasicAxisAlarms[E_BasicAxis.CommandWhileInhibited].Clear(0, 0);
END_IF

//ErrorID 16 - NC Axis Error
IF CamSlaveAxis.Axis.Status.Error AND NOT BasicAxisAlarms[E_BasicAxis.AxisError].bRaised THEN
	RaiseAlarmWithStrings(Alarm := BasicAxisAlarms[E_BasicAxis.AxisError], UDINT_TO_STRING(CamSlaveAxis.Axis.Status.ErrorID), '');
ELSIF NOT CamSlaveAxis.Axis.Status.Error AND BasicAxisAlarms[E_BasicAxis.AxisError].bRaised THEN
	BasicAxisAlarms[E_BasicAxis.AxisError].Clear(0, 0);
END_IF

//ErrorID 17 - Hardware Error **TODO**

//ErrorID 2 - MC_CamIn
IF CamSlaveAxis.McCamIn.Error AND NOT CamSlaveAxisAlarms[E_CamSlaveAxis.McCamInError].bRaised THEN
	RaiseAlarmWithStrings(Alarm := CamSlaveAxisAlarms[E_CamSlaveAxis.McCamInError], UDINT_TO_STRING(CamSlaveAxis.ErrorID), '');
ELSIF NOT CamSlaveAxis.McCamIn.Error AND CamSlaveAxisAlarms[E_CamSlaveAxis.McCamInError].bRaised THEN
	CamSlaveAxisAlarms[E_CamSlaveAxis.McCamInError].Clear(0, 0);
END_IF

//ErrorID 3 - MC_CamOut
IF CamSlaveAxis.McCamOut.Error AND NOT CamSlaveAxisAlarms[E_CamSlaveAxis.McCamOutError].bRaised THEN
	RaiseAlarmWithStrings(Alarm := CamSlaveAxisAlarms[E_CamSlaveAxis.McCamOutError], UDINT_TO_STRING(CamSlaveAxis.McCamOut.ErrorID), '');
ELSIF NOT CamSlaveAxis.McCamOut.Error AND CamSlaveAxisAlarms[E_CamSlaveAxis.McCamOutError].bRaised THEN
	CamSlaveAxisAlarms[E_CamSlaveAxis.McCamOutError].Clear(0, 0);
END_IF

//ErrorID 4 - MC_CamTableSelect
IF CamSlaveAxis.MCCamTableSelect.Error AND NOT CamSlaveAxisAlarms[E_CamSlaveAxis.McLoadCamTableError].bRaised THEN
	RaiseAlarmWithStrings(Alarm := CamSlaveAxisAlarms[E_CamSlaveAxis.McLoadCamTableError], UDINT_TO_STRING(CamSlaveAxis.MCCamTableSelect.ErrorID), '');
ELSIF NOT CamSlaveAxis.MCCamTableSelect.Error AND CamSlaveAxisAlarms[E_CamSlaveAxis.McLoadCamTableError].bRaised THEN
	CamSlaveAxisAlarms[E_CamSlaveAxis.McLoadCamTableError].Clear(0, 0);
END_IF

//ErrorID 5 - MC_ReadCamTableSlaveDynamics
IF CamSlaveAxis.MCReadCamTableSlaveDynamics.Error AND NOT CamSlaveAxisAlarms[E_CamSlaveAxis.McReadSlaveDynamicsError].bRaised THEN
	RaiseAlarmWithStrings(Alarm := CamSlaveAxisAlarms[E_CamSlaveAxis.McReadSlaveDynamicsError], UDINT_TO_STRING(CamSlaveAxis.MCReadCamTableSlaveDynamics.ErrorID), '');
ELSIF NOT CamSlaveAxis.MCReadCamTableSlaveDynamics.Error AND CamSlaveAxisAlarms[E_CamSlaveAxis.McReadSlaveDynamicsError].bRaised THEN
	CamSlaveAxisAlarms[E_CamSlaveAxis.McReadSlaveDynamicsError].Clear(0, 0);
END_IF

//ErrorID 6 - MC_SetCamOnlineChangeMode 
IF CamSlaveAxis.MCSetCamOnlineChangeMode.Error AND NOT CamSlaveAxisAlarms[E_CamSlaveAxis.McCamOnlineChangeModeError].bRaised THEN
	RaiseAlarmWithStrings(Alarm := CamSlaveAxisAlarms[E_CamSlaveAxis.McCamOnlineChangeModeError], UDINT_TO_STRING(CamSlaveAxis.MCSetCamOnlineChangeMode.ErrorID), '');
ELSIF NOT CamSlaveAxis.MCSetCamOnlineChangeMode.Error AND CamSlaveAxisAlarms[E_CamSlaveAxis.McCamOnlineChangeModeError].bRaised THEN
	CamSlaveAxisAlarms[E_CamSlaveAxis.McCamOnlineChangeModeError].Clear(0, 0);
END_IF

//ErrorID 7 - MC_WriteMotionFunction
IF CamSlaveAxis.McWriteMotionFunction.Error AND NOT CamSlaveAxisAlarms[E_CamSlaveAxis.McWriteMotionFunctionError].bRaised THEN
	RaiseAlarmWithStrings(Alarm := CamSlaveAxisAlarms[E_CamSlaveAxis.McWriteMotionFunctionError], UDINT_TO_STRING(CamSlaveAxis.McWriteMotionFunction.ErrorID), '');
ELSIF NOT CamSlaveAxis.McWriteMotionFunction.Error AND CamSlaveAxisAlarms[E_CamSlaveAxis.McWriteMotionFunctionError].bRaised THEN
	CamSlaveAxisAlarms[E_CamSlaveAxis.McWriteMotionFunctionError].Clear(0, 0);
END_IF

////ErrorID 8 - MC_ReadParameterSet

//IF CamSlaveAxis.McReadAxisParameters.Error AND NOT CamSlaveAxisAlarms[E_CamSlaveAxis.McReadAxisParametersError].bRaised THEN

//    RaiseAlarmWithStrings(Alarm := CamSlaveAxisAlarms[E_CamSlaveAxis.McReadAxisParametersError], UDINT_TO_STRING(CamSlaveAxis.McReadAxisParameters.ErrorID), '');

//ELSIF NOT CamSlaveAxis.McReadAxisParameters.Error AND CamSlaveAxisAlarms[E_CamSlaveAxis.McReadAxisParametersError].bRaised THEN

//    CamSlaveAxisAlarms[E_CamSlaveAxis.McReadAxisParametersError].Clear(0, 0);

//END_IF

//ErrorID 9 - CamControlSequenceError
IF CamSlaveAxis.SequenceError AND NOT CamSlaveAxisAlarms[E_CamSlaveAxis.CamControlSequenceError].bRaised THEN
	RaiseAlarmWithStrings(Alarm := CamSlaveAxisAlarms[E_CamSlaveAxis.CamControlSequenceError], UDINT_TO_STRING(CamSlaveAxis.SequenceErrorID), '');
ELSIF NOT CamSlaveAxis.SequenceError AND CamSlaveAxisAlarms[E_CamSlaveAxis.CamControlSequenceError].bRaised THEN
	CamSlaveAxisAlarms[E_CamSlaveAxis.CamControlSequenceError].Clear(0, 0);
END_IF

_CurrentAlarmSeverity := F_GetMaxSeverityRaised(Alarms := BasicAxisAlarms, CurrentSeverity := CurrentAlarmSeverity);
_CurrentAlarmSeverity := F_GetMaxSeverityRaised(Alarms := CamSlaveAxisAlarms, CurrentSeverity := CurrentAlarmSeverity);
END_METHOD

METHOD CyclicLogic
SUPER^.CyclicLogic();
CamSlaveAxis.CyclicLogic();
_Busy	 := CamSlaveAxis.Busy;
_Error	 := CamSlaveAxis.Error;
_ErrorID := CamSlaveAxis.ErrorID;
END_METHOD

//! @summary Basic component initialization logic
METHOD PROTECTED Initialize : BOOL;

//! @description This method is called by <c>CyclicLogic()</c> as required
IF NOT CamSlaveAxis.InitComplete THEN
	RETURN;
END_IF

Initialize := SUPER^.Initialize();
END_METHOD

END_FUNCTION_BLOCK

// Project Information/F_GetCompany
// This function has been automatically generated from the project information.
{attribute 'signature_flag' := '1073741824'}
{attribute 'TcGenerated'}
{attribute 'no-analysis'}
FUNCTION F_GetCompany : WSTRING
VAR_INPUT
	
END_VAR

F_GetCompany := "Beckhoff Automation LLC";

END_FUNCTION

// Project Information/F_GetTitle
// This function has been automatically generated from the project information.
{attribute 'signature_flag' := '1073741824'}
{attribute 'TcGenerated'}
{attribute 'no-analysis'}
FUNCTION F_GetTitle : WSTRING
VAR_INPUT
	
END_VAR

F_GetTitle := "SPT Components";

END_FUNCTION

// Project Information/F_GetVersion
// This function has been automatically generated from the project information.
{attribute 'signature_flag' := '1073741824'}
{attribute 'TcGenerated'}
{attribute 'no-analysis'}
FUNCTION F_GetVersion : ST_LibVersion
VAR_INPUT
	
END_VAR

F_GetVersion.iMajor := 3;
F_GetVersion.iMinor := 1;
F_GetVersion.iBuild := 1;
F_GetVersion.iRevision := 0;
F_GetVersion.sVersion := '3.1.1';
F_GetVersion.nFlags := 1;

END_FUNCTION

// Sensors/FB_DigitalSensor
FUNCTION_BLOCK FB_DigitalSensor EXTENDS FB_ComponentBase IMPLEMENTS I_DigitalSensorBase
VAR
	HardwareInput AT %I*		: BOOL;			  //Hardware input bit from the hysical sensor
	_DebounceMode				: E_DebounceMode; //Defines the debounce model that will filter the sensor's output to the program
	_DebounceTime				: TIME;			  //Time input parameter for use in Debounce functionality
	_Inverted					: BOOL;			  //Defines the output polarity of the sensor - a "TRUE" value will result in the signal of the sensor being inverted
	_SimulationInput			: BOOL;			  //Provides configuration input to the simulation functionality
	_SimulationTimebase			: UDINT;
	_SimulationMode				: E_SensorSimulationMode; //Defines the mode of operation for the simulation functionality of this component
	_TimeActive					: TIME;					  //Tracks the amount of time that the sensor has been in an active state
	_TimeInactive				: TIME;					  //Tracks the amount of time that the sensor has been in an inactive state
	_Active						: BOOL;
	TON_ActiveTimer				: Tc2_Standard.TON; //Tracks the amount of time that the sensor has been in an active state
	TON_InactiveTimer			: Tc2_Standard.TON; //Tracks the amount of time that the sensor has been in an inactive state
	TON_DebounceTimer			: Tc2_Standard.TON; //Utilized in the debounce implementation
	TP_DebounceTimer			: Tc2_Standard.TP;	//Utilized in the debounce implementation
	DigitalSensor_HMI			: ST_DigitalSensor_HMI;
	SimulationPulse1_TP			: Tc2_Standard.TP; //Pulse Timer for simulated sensor pulse generation
	SimulationPulse2_TP			: Tc2_Standard.TP; //Pulse Timer for simulated sensor pulse generation
	HMICommand_DigitalSensor_RT : R_TRIG;
END_VAR

METHOD PUBLIC CyclicLogic
VAR_INPUT
END_VAR
SUPER^.CyclicLogic();
IF _Simulate THEN
	CASE _SimulationMode OF
		E_SensorSimulationMode.InputDriven:
			_Active := _SimulationInput;

		E_SensorSimulationMode.Periodic:
			SimulationPulse1_TP(IN := NOT SimulationPulse2_TP.Q, PT := UDINT_TO_TIME(_SimulationTimebase));
			SimulationPulse2_TP(IN := NOT SimulationPulse1_TP.Q, PT := UDINT_TO_TIME(_SimulationTimebase));
			_Active := SimulationPulse2_TP.Q;
	END_CASE
ELSE
	_Active := ProcessInput(Input := HardwareInput);
END_IF
END_METHOD

PROPERTY Active : BOOL
GET
Active := _Active;
END_GET
END_PROPERTY

PROPERTY DebounceMode : E_DebounceMode
GET
DebounceMode := _DebounceMode;
END_GET
SET
_DebounceMode := DebounceMode;
END_SET
END_PROPERTY

PROPERTY DebounceTime : TIME
GET
DebounceTime := _DebounceTime;
END_GET
SET
_DebounceTime := DebounceTime;
END_SET
END_PROPERTY

PROPERTY Inverted : BOOL
GET
Inverted := _Inverted;
END_GET
SET
_Inverted := Inverted;
END_SET
END_PROPERTY

PROPERTY SimulationInput : BOOL
GET
SimulationInput := _SimulationInput;
END_GET
SET
_SimulationInput := SimulationInput;
END_SET
END_PROPERTY

PROPERTY SimulationMode : E_SensorSimulationMode
GET
SimulationMode := _SimulationMode;
END_GET
SET
_SimulationMode := SimulationMode;
END_SET
END_PROPERTY

PROPERTY SimulationTimeBase : UDINT
GET
SimulationTimeBase := _SimulationTimebase;
END_GET
SET
_SimulationTimeBase := SimulationTimebase;
END_SET
END_PROPERTY

PROPERTY TimeActive : TIME
GET
TimeActive := _TimeActive;
END_GET
END_PROPERTY

PROPERTY TimeInactive : TIME
GET
TimeInactive := _TimeInactive;
END_GET
END_PROPERTY

METHOD PROTECTED HMICommunication
//Extend this method in extended FBs to communicate specific implementation data
SUPER^.HMICommunication();

//Process HMI requests

//Replace 'FALSE' below with further momentary commands (myCommand XOR myOtherCommand XOR...)
HMICommand_DigitalSensor_RT(CLK := (ComponentBase_HMI.Status.HMIControlAvailable AND NOT HMICommandActive_Base) AND (FALSE));

//Signal to FB_ComponentBase that a command is active
HMICommandActive_Descendant := ComponentBase_HMI.Status.HMIControlAvailable AND
							   (DigitalSensor_HMI.Config.DebounceMode <> _DebounceMode OR DigitalSensor_HMI.Config.DebounceTime <> _DebounceTime OR DigitalSensor_HMI.Config.Inverted <> _Inverted OR
							   DigitalSensor_HMI.Config.SimulationMode <> _SimulationMode OR DigitalSensor_HMI.Config.SimulationTimebase <> _SimulationTimebase);

//Process HMI requests
IF HMICommand_DigitalSensor_RT.Q THEN //If a request has been issued by the HMI, and a previous request has not just finished being processed

	//	IF AxisBaseHMI.Command.xxx THEN

	//		Enabled := TRUE;

	//	END_IF
END_IF

IF ComponentBase_HMI.Status.HMIControlAvailable AND NOT HMICommand_DigitalSensor_RT.Q THEN
	IF DigitalSensor_HMI.Config.DebounceMode <> _DebounceMode THEN
		DebounceMode := DigitalSensor_HMI.Config.DebounceMode;
	END_IF

	IF DigitalSensor_HMI.Config.DebounceTime <> _DebounceTime THEN
		DebounceTime := DigitalSensor_HMI.Config.DebounceTime;
	END_IF

	IF DigitalSensor_HMI.Config.Inverted <> _Inverted THEN
		Inverted := DigitalSensor_HMI.Config.Inverted;
	END_IF

	IF DigitalSensor_HMI.Config.SimulationMode <> _SimulationMode THEN
		SimulationMode := DigitalSensor_HMI.Config.SimulationMode;
	END_IF

	IF DigitalSensor_HMI.Config.SimulationTimebase <> _SimulationTimebase THEN
		SimulationTimeBase := DigitalSensor_HMI.Config.SimulationTimebase;
	END_IF
END_IF

//Update HMI status info
DigitalSensor_HMI.Status.Active		  := _Active;
DigitalSensor_HMI.Status.TimeActive	  := TIME_TO_LREAL(_TimeActive) / 1000.0;
DigitalSensor_HMI.Status.TimeInactive := TIME_TO_LREAL(_TimeInactive) / 1000.0;
END_METHOD

METHOD PROTECTED Monitoring
SUPER^.Monitoring();

//If flicker counters or other diagnostic systems are desired, their implementation could be here

//Any warnings, errors, or other desired messages would also be generated here

//T#71582M47S295MS is the upper bound of the TIME type, meaning these timers will continue to increase ET for as long as possible
TON_ActiveTimer(IN := _Active, PT := T#71582M47S295MS, ET => _TimeActive);
TON_InactiveTimer(IN := NOT _Active, PT := T#71582M47S295MS, ET => _TimeInactive);
_Busy  := FALSE;
_Error := FALSE;
END_METHOD

METHOD PRIVATE ProcessInput : BOOL
VAR_INPUT
	Input : BOOL;
END_VAR

VAR
	DebouncedInput : BOOL;
END_VAR

VAR_INST
	LastDebouncedInput : BOOL;
	MovingAverage	   : DINT;
END_VAR
CASE DebounceMode OF
	E_DebounceMode.RawInput: //Passes raw input through
		DebouncedInput := Input;

	E_DebounceMode.SimpleFlickerFilter:											 //Requires the raw input to be a consistent value for a set time period before output changes
		TON_DebounceTimer(IN := (Input <> DebouncedInput), PT := _DebounceTime); //runs the timer whenever a differing input is detected
		IF TON_DebounceTimer.Q THEN
			DebouncedInput := Input; //once the raw input has been different for the specified debounce time, the processed input is updated
		END_IF

	E_DebounceMode.EdgeDetectFilter: //Updates the processed value immediately on a change from steady state, but mutes any sensor flickers for the specified time immediately following the change
		IF (Input <> DebouncedInput) AND (NOT TP_DebounceTimer.Q)
			THEN //A differing raw input must be detected outside of the mute window created by the pulse timer
			DebouncedInput := Input;
		END_IF

		TP_DebounceTimer(IN := (DebouncedInput <> LastDebouncedInput), PT := _DebounceTime); //"Q" will be TRUE for tDebounce time after the bProcessedSensorInput value is changed
	E_DebounceMode.MovingAverage
		: //Uses a "moving average"-like calculation to compensate for extremely inconsistent signals - prevents poorly timed flickers from causing disproportionate results
		TON_DebounceTimer(IN := NOT TON_DebounceTimer.Q,
						  PT := T#5MS); //Provides a 1ms "polling" trigger

		IF TON_DebounceTimer.Q THEN									//TRUE once every millisecond
			IF Input THEN											//If raw input is currently active at the time of polling
				IF MovingAverage < TIME_TO_DINT(_DebounceTime) THEN //If the moving average has not reached its "weight limit" as set by debounce time
					MovingAverage := MovingAverage + 5;				//Add 1 to the average
				END_IF
			ELSE													 //If raw input is currently inactive at the time of polling
				IF MovingAverage > -TIME_TO_DINT(_DebounceTime) THEN //If the moving average has not reached its "weight limit" as set by debounce time
					MovingAverage := MovingAverage - 5;				 //Subtract 1 from the average
				END_IF
			END_IF
		END_IF

		IF MovingAverage >= 0 THEN
			DebouncedInput := TRUE;
		ELSE
			DebouncedInput := FALSE;
		END_IF
END_CASE

LastDebouncedInput := DebouncedInput; //Update "Last value"
IF _Inverted THEN					  //If signal inversion is requested, invert the signal
	DebouncedInput := NOT DebouncedInput;
END_IF

ProcessInput := DebouncedInput;
END_METHOD

END_FUNCTION_BLOCK

// Sensors/I_DigitalSensorBase
INTERFACE I_DigitalSensorBase

PROPERTY DebounceMode : E_DebounceMode
GET
END_GET
SET
END_SET
END_PROPERTY

PROPERTY DebounceTime : TIME
GET
END_GET
SET
END_SET
END_PROPERTY

PROPERTY Inverted : BOOL //"High" signal from the sensor will be interpreted as an "inactive" reading when this parameter is TRUE
GET
END_GET
SET
END_SET
END_PROPERTY

PROPERTY SimulationInput : BOOL
GET
END_GET
SET
END_SET
END_PROPERTY

PROPERTY SimulationMode : E_SensorSimulationMode
GET
END_GET
SET
END_SET
END_PROPERTY

PROPERTY TimeActive : TIME
GET
END_GET
END_PROPERTY

PROPERTY TimeInactive : TIME
GET
END_GET
END_PROPERTY

END_INTERFACE

// Solenoids/SolenoidBankBase/FB_SolenoidBankBase
FUNCTION_BLOCK ABSTRACT FB_SolenoidBankBase EXTENDS FB_ComponentBase
VAR
	// Configuration
	Configuration : ARRAY[1..Parameters_Cylinder.MAX_NUMBER_OF_SOLENOIDS] OF ST_SolenoidBankConfig;

	//Counted number of solenoids
	NumberOfSolenoids : UINT;

	//Alarms
	SolenoidBankAlarms : ARRAY[1..SolenoidBankBaseAlarmsCount] OF FB_TcAlarm;
END_VAR

VAR CONSTANT
	SolenoidBankBaseAlarmsCount : UINT := 2;
END_VAR

METHOD PUBLIC AddSolenoid : UINT
VAR_INPUT
	ipCylinder	 : I_Solenoid;
	Number		 : UINT; //This is the number in the IO tree.
	SolenoidType : E_SolenoidType;
END_VAR
IF CheckNumber(Number) AND ipCylinder <> 0 THEN
	NumberOfSolenoids									  := NumberOfSolenoids + 1;
	Configuration[NumberOfSolenoids].ipSolenoid			  := ipCylinder;
	Configuration[NumberOfSolenoids].SolenoidType		  := SolenoidType;
	Configuration[NumberOfSolenoids].SolenoidOutputNumber := Number;
END_IF
END_METHOD

METHOD PRIVATE CheckNumber : BOOL
VAR_INPUT
	Number : UINT;
END_VAR
CheckNumber := TRUE;
IF Number < 1 AND Number > Parameters_Cylinder.MAX_NUMBER_OF_SOLENOIDS THEN
	IF NOT SolenoidBankAlarms[E_CylinderBankAlarms.CylinderNumberOutOfRange].bRaised THEN
		SolenoidBankAlarms[E_CylinderBankAlarms.CylinderNumberOutOfRange].Raise(0);
	END_IF

	CheckNumber := FALSE;
END_IF
END_METHOD

//! @summary Initializes event function blocks using this components's name
{attribute 'call_after_online_change_slot' := '<slot>'}
METHOD PROTECTED CreateEvents

//! @description This method is called by <c>Initialize()</c> as required
SUPER^.CreateEvents();
F_CreateAllEventsInClass(Alarms		:= SolenoidBankAlarms,
						 ClassSize	:= SIZEOF(TC_EVENTS.CylinderBankAlarms),
						 pInitEvent := ADR(TC_EVENTS.CylinderBankAlarms.InitReferenceEvent),
						 Prefix		:= Name);
END_METHOD

//! @summary This method serves as the entry point for all underlying FB logic
METHOD PUBLIC CyclicLogic
//! @description This method should be called cyclically by descendant function blocks by invoking <c>SUPER^.CyclicLogic()</c>.  Alternatively, the contents of this method could be reimplemented entirely in which case a call to this method would not be necessary.
VAR
	x : UINT;
END_VAR
//Loop through all solenoids that are added.
FOR x := 1 TO NumberOfSolenoids DO
	MapIO(x);
END_FOR
END_METHOD

//! @summary Basic component initialization logic
METHOD PROTECTED Initialize : BOOL;
//! @description This method is called by <c>CyclicLogic()</c> as required
VAR
	x : UINT;
END_VAR
NumberOfSolenoids := 0;
Initialize		  := TRUE;
END_METHOD

METHOD ABSTRACT MapIO
VAR_INPUT
	x : UINT;
END_VAR
END_METHOD

//! Provides basic error detection and event handling for this component
METHOD PROTECTED Monitoring

(*! @descriptionThis method is called cyclically by <c>CyclicLogic()</c>*)
SUPER^.Monitoring();
_CurrentAlarmSeverity := F_GetMaxSeverityRaised(Alarms := SolenoidBankAlarms, CurrentSeverity := CurrentAlarmSeverity);
END_METHOD

//! @summary Clears error flags and error IDs for this component
METHOD PUBLIC Reset : BOOL
SUPER^.Reset();
IF SolenoidBankAlarms[E_CylinderBankAlarms.CylinderNumberOutOfRange].bRaised THEN
	SolenoidBankAlarms[E_CylinderBankAlarms.CylinderNumberOutOfRange].Clear(0, 0);
END_IF
END_METHOD

END_FUNCTION_BLOCK

// Solenoids/I_Solenoid
INTERFACE I_Solenoid

METHOD Extend
VAR_INPUT
END_VAR
END_METHOD

PROPERTY Extended : BOOL
GET
END_GET
END_PROPERTY

PROPERTY ExtendOutput : BOOL
GET
END_GET
END_PROPERTY

PROPERTY ExtendTime : LREAL
GET
END_GET
SET
END_SET
END_PROPERTY

METHOD Retract
VAR_INPUT
END_VAR
END_METHOD

PROPERTY Retracted : BOOL
GET
END_GET
END_PROPERTY

PROPERTY RetractOutput : BOOL
GET
END_GET
END_PROPERTY

PROPERTY RetractTime : LREAL
GET
END_GET
SET
END_SET
END_PROPERTY

END_INTERFACE

// Solenoids/FB_DoubleSolenoid
FUNCTION_BLOCK FB_DoubleSolenoid EXTENDS FB_SingleSolenoid
VAR
	_RetractOutput AT %Q* : BOOL;
END_VAR

METHOD PROTECTED HardwareInit
//Update the status based on the IO 
IF _ExtendOutput AND NOT _RetractOutput THEN
	_Extended  := TRUE;
	_Retracted := FALSE;
ELSIF NOT _ExtendOutput AND _RetractOutput THEN
	_Extended  := FALSE;
	_Retracted := TRUE;
ELSE // By Default, set RetractOuptupt if neither is set or if both are set.
	_ExtendOutput  := FALSE;
	_RetractOutput := TRUE;
	_Extended	   := FALSE;
	_Retracted	   := TRUE;
END_IF
END_METHOD

METHOD PROTECTED HardwareUpdate
//One shot the requests
Extend_RTRIG(CLK := _ExtendRequest);
Retract_RTRIG(CLK := _RetractRequest);

//Handle Extend
IF Extend_RTRIG.Q THEN
	_ExtendOutput	:= TRUE;
	_RetractOutput	:= FALSE;
	_Extending		:= TRUE;
	_Retracting		:= FALSE;
	_Retracted		:= FALSE;
	_RetractRequest := FALSE;
END_IF

//Handle Retract
IF Retract_RTRIG.Q THEN
	_ExtendOutput  := FALSE;
	_RetractOutput := TRUE;
	_Extending	   := FALSE;
	_Retracting	   := TRUE;
	_Extended	   := FALSE;
	_ExtendRequest := FALSE;
END_IF

//Always Simulate Feedback here with no feedback inputs
Feedback();
END_METHOD

PROPERTY RetractOutput : BOOL
GET
RetractOutput := _RetractOutput;
END_GET
END_PROPERTY

END_FUNCTION_BLOCK

// Solenoids/FB_SingleSolenoid
(*	This FB is used for a single output solenoid 
	It uses the times to say when Extended/Retracted  	
	It starts assuming retracted and the output off.
*)
FUNCTION_BLOCK FB_SingleSolenoid EXTENDS FB_ComponentBase IMPLEMENTS I_Solenoid
VAR
	//Output
	_ExtendOutput AT %Q* : BOOL;

	// Internal variables
	_ExtendRequest	: BOOL;
	_RetractRequest : BOOL;
	_Extended		: BOOL;
	_Retracted		: BOOL;
	_Extending		: BOOL;
	_Retracting		: BOOL;
	_ExtendTime		: LREAL := 1000; // Default time 1s
	_RetractTime	: LREAL := 1000; // Default time 1s

	// Timer for Extend/Retract
	Extend_TON	  : TON;
	Retract_TON	  : TON;
	Extend_RTRIG  : R_TRIG;
	Retract_RTRIG : R_TRIG;

	//HMI 
	SolenoidHMI : ST_Cylinder_HMI;

	//Alarms
	SolenoidAlarms : ARRAY[1..SolenoidAlarmsCount] OF FB_TcAlarm;
END_VAR

VAR CONSTANT
	SolenoidAlarmsCount : UINT := 4;
END_VAR

METHOD PROTECTED CreateEvents
VAR_INPUT
END_VAR
SUPER^.CreateEvents();
F_CreateAllEventsInClass(Alarms		:= SolenoidAlarms,
						 ClassSize	:= SIZEOF(TC_EVENTS.CylinderAlarms),
						 pInitEvent := ADR(TC_EVENTS.CylinderAlarms.InitReferenceEvent),
						 Prefix		:= Name);
END_METHOD

METHOD PROTECTED HMICommunication
VAR_INPUT
END_VAR
SUPER^.HMICommunication();

//Handle the requests to extend and retract
IF ComponentBase_HMI.Status.HMIControlAvailable THEN
	IF SolenoidHMI.Command.Extend THEN
		Extend();
	ELSIF SolenoidHMI.Command.Retract THEN
		Retract();
	END_IF

	IF NOT F_CompareLREAL(SolenoidHMI.Command.ExtendTime, _ExtendTime, 0.01) THEN
		_ExtendTime := SolenoidHMI.Command.ExtendTime;
	END_IF

	IF NOT F_CompareLREAL(SolenoidHMI.Command.RetractTime, _RetractTime, 0.01) THEN
		_RetractTime := SolenoidHMI.Command.RetractTime;
	END_IF
END_IF

//Update HMI status info
SolenoidHMI.Status.Extended	   := _Extended;
SolenoidHMI.Status.Extending   := _Extending;
SolenoidHMI.Status.Retracted   := _Retracted;
SolenoidHMI.Status.Retracting  := _Retracting;
SolenoidHMI.Config.ExtendTime  := _ExtendTime;
SolenoidHMI.Config.RetractTime := _RetractTime;
END_METHOD

METHOD PROTECTED Monitoring
VAR_INPUT
END_VAR
SUPER^.Monitoring();

//Update output bits
_Busy				  := _Extending OR _Retracting;
_CurrentAlarmSeverity := F_GetMaxSeverityRaised(Alarms := SolenoidAlarms, CurrentSeverity := CurrentAlarmSeverity);
_Error				  := _CurrentAlarmSeverity >= TcEventSeverity.Error;
END_METHOD

METHOD CyclicLogic
VAR
	myErrorID : UDINT;
END_VAR
HardwareUpdate();
SUPER^.CyclicLogic();

//New code
myErrorID := THIS^.ErrorID;
END_METHOD

METHOD Extend
_ExtendRequest	:= TRUE;
_RetractRequest := FALSE;
END_METHOD

PROPERTY Extended : BOOL
GET
Extended := _Extended;
END_GET
END_PROPERTY

PROPERTY ExtendOutput : BOOL
GET
ExtendOutput := _ExtendOutput;
END_GET
END_PROPERTY

PROPERTY ExtendTime : LREAL
GET
ExtendTime := _ExtendTime;
END_GET
SET
_ExtendTime					   := ExtendTime;
SolenoidHMI.Command.ExtendTime := ExtendTime;
END_SET
END_PROPERTY

METHOD Retract
_ExtendRequest	:= FALSE;
_RetractRequest := TRUE;
END_METHOD

PROPERTY Retracted : BOOL
GET
Retracted := _Retracted;
END_GET
END_PROPERTY

PROPERTY RetractOutput : BOOL
GET
RetractOutput := FALSE;
END_GET
END_PROPERTY

PROPERTY RetractTime : LREAL
GET
RetractTime := _RetractTime;
END_GET
SET
_RetractTime					:= RetractTime;
SolenoidHMI.Command.RetractTime := RetractTime;
END_SET
END_PROPERTY

METHOD PROTECTED Feedback
VAR_INPUT
END_VAR
//Handle the time to Extend/Retract
Extend_TON(IN := _Extending, PT := LREAL_TO_TIME(_ExtendTime));
Retract_TON(IN := _Retracting, PT := LREAL_TO_TIME(_RetractTime));
IF Extend_TON.Q THEN
	_Extended  := TRUE;
	_Extending := FALSE;
END_IF

IF Retract_TON.Q THEN
	_Retracted	:= TRUE;
	_Retracting := FALSE;
END_IF
END_METHOD

METHOD PROTECTED HardwareInit
IF _ExtendOutput THEN
	_Extended  := TRUE;
	_Retracted := FALSE;
ELSE
	_Extended  := FALSE;
	_Retracted := TRUE;
END_IF
END_METHOD

METHOD PROTECTED HardwareUpdate
VAR_INPUT
END_VAR
//One shot the requests
Extend_RTRIG(CLK := _ExtendRequest);
Retract_RTRIG(CLK := _RetractRequest);

//Handle Extend
IF Extend_RTRIG.Q THEN
	_ExtendOutput	:= TRUE;
	_Extending		:= TRUE;
	_Retracting		:= FALSE;
	_Retracted		:= FALSE;
	_RetractRequest := FALSE;
END_IF

//Handle Retract
IF Retract_RTRIG.Q THEN
	_ExtendOutput  := FALSE;
	_Extending	   := FALSE;
	_Retracting	   := TRUE;
	_Extended	   := FALSE;
	_ExtendRequest := FALSE;
END_IF

//Call the feedback 
Feedback();
END_METHOD

//! @summary Basic component initialization logic
METHOD PROTECTED Initialize : BOOL;

//! @description This method is called by <c>CyclicLogic()</c> as required
//Set the cylinder to retracted
_Extending		:= FALSE;
_ExtendRequest	:= FALSE;
_Retracting		:= FALSE;
_RetractRequest := FALSE;

//Set the HMI time to the currnt time.
SolenoidHMI.Command.ExtendTime	:= _ExtendTime;
SolenoidHMI.Command.RetractTime := _RetractTime;

//Call base class Initialize
Initialize := SUPER^.Initialize();

// Call the HardwareInit
HardwareInit();
END_METHOD

//! @summary Clears error flags and error IDs for this component
METHOD PUBLIC Reset : BOOL
Reset := FALSE;
F_ClearAllEventsInClass(Alarms := SolenoidAlarms);
END_METHOD

END_FUNCTION_BLOCK

// Solenoids/FB_DoubleSolenoidFeedback
FUNCTION_BLOCK FB_DoubleSolenoidFeedback EXTENDS FB_DoubleSolenoid
VAR
	ExtendedSensor	AT %I* : BOOL;
	RetractedSensor AT %I* : BOOL;
END_VAR

PROPERTY ExtendedInput : BOOL
SET
ExtendedSensor := ExtendedInput;
END_SET
END_PROPERTY

METHOD PROTECTED Feedback
IF NOT _Simulate THEN
	_Extended  := ExtendedSensor;
	_Retracted := RetractedSensor;
	Extend_TON(IN := _Extending, PT := LREAL_TO_TIME(_ExtendTime));
	Retract_TON(IN := _Retracting, PT := LREAL_TO_TIME(_RetractTime));
	IF Extend_TON.Q AND NOT ExtendedSensor THEN
		IF NOT SolenoidAlarms[E_CylinderAlarms.ExtendTimeout].bRaised THEN
			SolenoidAlarms[E_CylinderAlarms.ExtendTimeout].Raise(0);
			_ExtendRequest := FALSE;
			_Extending	   := FALSE;
		END_IF
	ELSIF _Extending AND ExtendedSensor THEN
		_Extended  := TRUE;
		_Extending := FALSE;
	END_IF

	IF Retract_TON.Q AND NOT RetractedSensor THEN
		IF NOT SolenoidAlarms[E_CylinderAlarms.RetractTimeout].bRaised THEN
			SolenoidAlarms[E_CylinderAlarms.RetractTimeout].Raise(0);
			_RetractRequest := FALSE;
			_Retracting		:= FALSE;
		END_IF
	ELSIF _Retracting AND RetractedSensor THEN
		_Retracted	:= TRUE;
		_Retracting := FALSE;
	END_IF
ELSE
	SUPER^.Feedback();
END_IF

//Monitor Inputs in case both on at the same time
IF ExtendedSensor AND RetractedSensor AND NOT SolenoidAlarms[E_CylinderAlarms.ExtendedAndRetracted].bRaised THEN
	SolenoidAlarms[E_CylinderAlarms.ExtendedAndRetracted].Raise(0);
ELSIF (ExtendedSensor XOR RetractedSensor) AND SolenoidAlarms[E_CylinderAlarms.ExtendedAndRetracted].bRaised THEN
	SolenoidAlarms[E_CylinderAlarms.ExtendedAndRetracted].Clear(0, 0);
END_IF
END_METHOD

METHOD PROTECTED HardwareInit
IF ExtendedSensor AND NOT RetractedSensor THEN
	_Extended  := TRUE;
	_Retracted := FALSE;
ELSIF NOT ExtendedSensor AND RetractedSensor THEN
	_Extended  := FALSE;
	_Retracted := TRUE;
ELSE // With Neither on, then this means that it is not either or maybe no air
	_Extended  := FALSE;
	_Retracted := FALSE;
END_IF
END_METHOD

PROPERTY RetractedInput : BOOL
SET
RetractedSensor := RetractedInput;
END_SET
END_PROPERTY

END_FUNCTION_BLOCK

// Solenoids/FB_SingleSolenoidFeedback
FUNCTION_BLOCK FB_SingleSolenoidFeedback EXTENDS FB_SingleSolenoid
VAR
	ExtendedSensor	AT %I* : BOOL;
	RetractedSensor AT %I* : BOOL;
END_VAR

PROPERTY ExtendedInput : BOOL
SET
ExtendedSensor := ExtendedInput;
END_SET
END_PROPERTY

METHOD PROTECTED Feedback
IF NOT _Simulate THEN
	_Extended  := ExtendedSensor;
	_Retracted := RetractedSensor;
	Extend_TON(IN := _Extending, PT := LREAL_TO_TIME(_ExtendTime));
	Retract_TON(IN := _Retracting, PT := LREAL_TO_TIME(_RetractTime));
	IF Extend_TON.Q AND NOT ExtendedSensor THEN
		IF NOT SolenoidAlarms[E_CylinderAlarms.ExtendTimeout].bRaised THEN
			SolenoidAlarms[E_CylinderAlarms.ExtendTimeout].Raise(0);
			_ExtendRequest := FALSE;
			_Extending	   := FALSE;
		END_IF
	ELSIF _Extending AND ExtendedSensor THEN
		_Extended  := TRUE;
		_Extending := FALSE;
	END_IF

	IF Retract_TON.Q AND NOT RetractedSensor THEN
		IF NOT SolenoidAlarms[E_CylinderAlarms.RetractTimeout].bRaised THEN
			SolenoidAlarms[E_CylinderAlarms.RetractTimeout].Raise(0);
			_RetractRequest := FALSE;
			_Retracting		:= FALSE;
		END_IF
	ELSIF _Retracting AND RetractedSensor THEN
		_Retracted	:= TRUE;
		_Retracting := FALSE;
	END_IF
ELSE
	SUPER^.Feedback(); //Call the feedback that usese timers for feedback
END_IF

//Monitor Inputs in case both on at the same time
IF ExtendedSensor AND RetractedSensor AND NOT SolenoidAlarms[E_CylinderAlarms.ExtendedAndRetracted].bRaised THEN
	SolenoidAlarms[E_CylinderAlarms.ExtendedAndRetracted].Raise(0);
ELSIF (ExtendedSensor XOR RetractedSensor) AND SolenoidAlarms[E_CylinderAlarms.ExtendedAndRetracted].bRaised THEN
	SolenoidAlarms[E_CylinderAlarms.ExtendedAndRetracted].Clear(0, 0);
END_IF
END_METHOD

METHOD PROTECTED HardwareInit
IF ExtendedSensor AND NOT RetractedSensor THEN
	_Extended  := TRUE;
	_Retracted := FALSE;
ELSIF NOT ExtendedSensor AND RetractedSensor THEN
	_Extended  := FALSE;
	_Retracted := TRUE;
ELSE // With Neither on, then this means that it is not either or maybe no air
	_Extended  := FALSE;
	_Retracted := FALSE;
END_IF
END_METHOD

PROPERTY RetractedInput : BOOL
SET
RetractedSensor := RetractedInput;
END_SET
END_PROPERTY

END_FUNCTION_BLOCK

// Testing/Axis/FB_ComponentBasicAxis_Test
FUNCTION_BLOCK FB_ComponentBasicAxis_Test EXTENDS TCUnit.FB_TestSuite
VAR
	TestFBInit					: FB_Component_BasicAxis;
	TestFBNameSetProperty		: FB_Component_BasicAxis;
	TestFBSimulationSetProperty : FB_Component_BasicAxis;
	TestFBSimulationSetHMI		: FB_Component_BasicAxis;
	TestFBSimulationCheckAlarm	: FB_Component_BasicAxis;
	TestFBBusy					: FB_Component_BasicAxis;
	TestFBAllowHMI				: FB_Component_BasicAxis;
	TestFBBlockHMI				: FB_Component_BasicAxis;

	//Axis integration test - this should be tested in the NCAxis library. (Enable, Disable, etc....)

	//Alarm Testing - 17 Alarms with FB_ComponentBasicAxis

	///TestFBAlarm1  FB_Component_BasicAxis; // InitReference (Not an actual alarm)
	TestFBAlarm2 : FB_Component_BasicAxis; // MC_Power
	TestFBAlarm3 : FB_Component_BasicAxis; // MC_Reset
	TestFBAlarm4 : FB_Component_BasicAxis; // MC_Halt

	///TestFBAlarm5 FB_Component_BasicAxis; // MC_Stop // Not Implemented
	TestFBAlarm6  : FB_Component_BasicAxis; // MC_Home
	TestFBAlarm7  : FB_Component_BasicAxis; // MC_Jog
	TestFBAlarm8  : FB_Component_BasicAxis; // MC_MoveAbsolute
	TestFBAlarm9  : FB_Component_BasicAxis; // MC_MoveRelative
	TestFBAlarm10 : FB_Component_BasicAxis; // MC_MoveVelocity
	TestFBAlarm11 : FB_Component_BasicAxis; // MC_MoveModulo
	TestFBAlarm12 : FB_Component_BasicAxis; // MC_ReadParameter
	TestFBAlarm13 : FB_Component_BasicAxis; // MC_WriteParameter
	TestFBAlarm14 : FB_Component_BasicAxis; // MC_WriteBOOLParameter
	TestFBAlarm15 : FB_Component_BasicAxis; // Command While Inhibited

	///TestFBAlarm16 FB_Component_BasicAxis; // Axis Error (Not Sure how to get Axis error with virtual axis)

	///TestFBAlarm17 FB_Component_BasicAxis; // Drive Error (Cannot Get Drive Error without drive)
END_VAR

Init();
NameSetProperty();
SimulationSetProperty();
SimulationSetHMI();
SimulationCheckAlarm();
Busy();
AllowHMI();
BlockHMI();

//Tests for Alarms
MCPowerAlarm();
MCResetAlarm();
MCHaltAlarm();
MCHomeAlarm();
MCJogAlarm();
MCMoveAbsoluteAlarm();
MCMoveRelativeAlarm();
MCMoveVelocity();
MCMoveModulo();
McReadAxisParametersAlarm();
McWriteAxisParameterAlarm();
McWriteAxisBoolParameterAlarm();
CommandInhibited();

METHOD AllowHMI
VAR_INST
	State		   : INT;
	ActualResult   : BOOL;
	ExpectedResult : BOOL := TRUE;
END_VAR
IF TEST_ORDERED('BasicAxisAllowHMI') THEN
	CASE State OF
		0:
			State := State + 10;

		10:
			IF TestFBAllowHMI.InitComplete AND NOT TestFBAllowHMI.Busy THEN
				TestFBAllowHMI.AllowHMIControl();
				State := State + 10;
			END_IF

		20:
			ActualResult := TestFBAllowHMI.ComponentBase_HMI.Status.HMIControlAvailable;
			AssertEquals_BOOL(Expected := ExpectedResult, Actual := ActualResult, Message := 'Function Block read allow HMI Control in HMI Tag not true');
			TEST_FINISHED();
			State := State + 10;
	END_CASE

	//Call to FB Cyclic Logic
	TestFBAllowHMI.CyclicLogic();
END_IF
END_METHOD

METHOD BlockHMI
VAR_INST
	State		   : INT;
	ActualResult   : BOOL;
	ExpectedResult : BOOL := FALSE;
END_VAR
IF TEST_ORDERED('BasicAxisBlockHMI') THEN
	CASE State OF
		0:
			State := State + 10;

		10:
			IF TestFBBlockHMI.InitComplete AND NOT TestFBBlockHMI.Busy THEN
				TestFBBlockHMI.AllowHMIControl();
				State := State + 10;
			END_IF

		20:
			IF TestFBBlockHMI.ComponentBase_HMI.Status.HMIControlAvailable THEN
				TestFBBlockHMI.BlockHMIControl();
				State := State + 10;
			END_IF

		30:
			ActualResult := TestFBBlockHMI.ComponentBase_HMI.Status.HMIControlAvailable;
			AssertEquals_BOOL(Expected := ExpectedResult, Actual := ActualResult, Message := 'Function Block read Block HMI Control in HMI Tag not false');
			TEST_FINISHED();
			State := State + 10;
	END_CASE

	//Call to FB Cyclic Logic
	TestFBBlockHMI.CyclicLogic();
END_IF
END_METHOD

METHOD Busy
VAR_INST
	State		   : INT;
	ActualResult   : BOOL;
	ExpectedResult : BOOL := TRUE;
	Timeout		   : TON;
END_VAR
IF TEST_ORDERED('BasicAxisBusy') THEN
	CASE State OF
		0:
			State := State + 10;

		10:
			IF TestFBBusy.InitComplete AND NOT TestFBBusy.Busy THEN
				TestFBBusy.Enable();
				State := State + 10;
			END_IF

		20:
			IF TestFBBusy.Enabled THEN
				TestFBBusy.Acceleration := 1000;
				TestFBBusy.Deceleration := 1000;
				TestFBBusy.Velocity		:= 100;
				TestFBBusy.MoveAbsolute(100, TRUE);
				State := State + 10;
			END_IF

		30:
			ActualResult := TestFBBusy.Busy;
			AssertEquals_BOOL(Expected := ExpectedResult, Actual := ActualResult, Message := 'Function Block was not busy when Extending');
			TEST_FINISHED();
			State := State + 10;
	END_CASE

	//Call to FB Cyclic Logic
	TestFBBusy.CyclicLogic();
END_IF
END_METHOD

METHOD CommandInhibited
VAR_INST
	State		   : INT;
	ActualResult   : BOOL;
	ExpectedResult : BOOL := TRUE;
END_VAR
IF TEST_ORDERED('CommandInhibitedAlarm') THEN
	CASE State OF
		0:
			IF TestFBAlarm15.InitComplete THEN
				TestFBAlarm15.Override := 0;
				TestFBAlarm15.MoveAbsolute(100, TRUE);
				State := State + 10;
			END_IF

		10:
			IF TestFBAlarm15.Error OR (TestFBAlarm15.InPosition AND NOT TestFBAlarm15.Busy) THEN
				ActualResult := TestFBAlarm15.BasicAxisAlarms[E_BasicAxis.CommandWhileInhibited].bRaised;
				State		 := State + 10;
			END_IF

		20:
			AssertEquals_BOOL(Expected := ExpectedResult, Actual := ActualResult, Message := 'The alarm was not raised for Command Inhibited Error');
			TEST_FINISHED();
			State := State + 10;
	END_CASE

	TestFBAlarm15.CyclicLogic();
END_IF
END_METHOD

METHOD Init
VAR_INST
	State		   : INT;
	ActualResult   : BOOL;
	ExpectedResult : BOOL := TRUE;
	Timeout		   : TON;
END_VAR
IF TEST_ORDERED('BasicAxisInit') THEN
	CASE State OF
		0:
			Timeout.IN := TRUE;
			State	   := State + 10;

		10:
			IF TestFBInit.InitComplete AND NOT TestFBInit.Busy THEN
				State := State + 10;
			END_IF

			IF Timeout.Q THEN
				State := State + 10;
			END_IF

		20:
			ActualResult := TestFBInit.InitComplete;
			AssertEquals_BOOL(Expected := ExpectedResult, Actual := ActualResult, Message := 'Function Block did not init complete in 2s');
			TEST_FINISHED();
			State := State + 10;
	END_CASE

	//Call to FB Cyclic Logic
	Timeout(PT := T#2S);
	TestFBInit.CyclicLogic();
END_IF
END_METHOD

METHOD MCHaltAlarm
VAR_INST
	State		   : INT;
	ActualResult   : BOOL;
	ExpectedResult : BOOL := TRUE;
	WriteADS	   : FB_WriteAdsSymByName;
END_VAR
IF TEST_ORDERED('MCHaltAlarm') THEN
	CASE State OF
		0:
			WriteADS(bWrite	  := TRUE,
					 sNetId	  := '',
					 nPort	  := 851,
					 sVarName := 'PRG_TEST.ComponentBasicAxisTest.TestFBAlarm4.BasicAxis.MCHalt.Error',
					 nSrcAddr := ADR(ExpectedResult),
					 nLen	  := SIZEOF(ExpectedResult),
					 tTimeout := T#2S,
					 eComMode :=,
					 bBusy	  =>,
					 bError	  =>,
					 nErrorId =>);

			IF NOT WriteADS.bBusy OR WriteADS.bError THEN
				State := State + 10;
			END_IF

			IF TestFBAlarm4.BasicAxisAlarms[E_BasicAxis.HaltError].bRaised THEN
				ActualResult := TestFBAlarm4.BasicAxisAlarms[E_BasicAxis.HaltError].bRaised;
				State		 := State + 10;
			END_IF

		10:
			AssertEquals_BOOL(Expected := ExpectedResult, Actual := ActualResult, Message := 'The alarm was not raised for MC_Halt.Error');
			TEST_FINISHED();
			State := State + 10;
	END_CASE

	TestFBAlarm4.CyclicLogic();
END_IF
END_METHOD

METHOD MCHomeAlarm
VAR_INST
	State		   : INT;
	ActualResult   : BOOL;
	ExpectedResult : BOOL := TRUE;
	WriteADS	   : FB_WriteAdsSymByName;
END_VAR
IF TEST_ORDERED('MCHomeAlarm') THEN
	CASE State OF
		0:
			WriteADS(bWrite	  := TRUE,
					 sNetId	  := '',
					 nPort	  := 851,
					 sVarName := 'PRG_TEST.ComponentBasicAxisTest.TestFBAlarm6.BasicAxis.DefaultHome._Error',
					 nSrcAddr := ADR(ExpectedResult),
					 nLen	  := SIZEOF(ExpectedResult),
					 tTimeout := T#2S,
					 eComMode :=,
					 bBusy	  =>,
					 bError	  =>,
					 nErrorId =>);

			IF NOT WriteADS.bBusy OR WriteADS.bError THEN
				State := State + 10;
			END_IF

			IF TestFBAlarm6.BasicAxisAlarms[E_BasicAxis.HomeError].bRaised THEN
				ActualResult := TestFBAlarm6.BasicAxisAlarms[E_BasicAxis.HomeError].bRaised;
				State		 := State + 10;
			END_IF

		10:
			AssertEquals_BOOL(Expected := ExpectedResult, Actual := ActualResult, Message := 'The alarm was not raised for HomeMethod.Error');
			TEST_FINISHED();
			State := State + 10;
	END_CASE

	TestFBAlarm6.CyclicLogic();
END_IF
END_METHOD

METHOD MCJogAlarm
VAR_INST
	State		   : INT;
	ActualResult   : BOOL;
	ExpectedResult : BOOL := TRUE;
	WriteADS	   : FB_WriteAdsSymByName;
END_VAR
IF TEST_ORDERED('MCJogAlarm') THEN
	CASE State OF
		0:
			WriteADS(bWrite	  := TRUE,
					 sNetId	  := '',
					 nPort	  := 851,
					 sVarName := 'PRG_TEST.ComponentBasicAxisTest.TestFBAlarm7.BasicAxis.MCJog.Error',
					 nSrcAddr := ADR(ExpectedResult),
					 nLen	  := SIZEOF(ExpectedResult),
					 tTimeout := T#2S,
					 eComMode :=,
					 bBusy	  =>,
					 bError	  =>,
					 nErrorId =>);

			IF NOT WriteADS.bBusy OR WriteADS.bError THEN
				State := State + 10;
			END_IF

			IF TestFBAlarm7.BasicAxisAlarms[E_BasicAxis.JogError].bRaised THEN
				ActualResult := TestFBAlarm7.BasicAxisAlarms[E_BasicAxis.JogError].bRaised;
				State		 := State + 10;
			END_IF

